// TwinCAT 3 PLC project Plc
// ProgramVersion: 3.1.4024.0
// libraries:
//   CHALET_BaseComponents, * (Beckhoff CH)
//   CHALET_Nc, * (Beckhoff CH)
//   CHALET_Xts, * (Beckhoff CH)
//   Tc2_ControllerToolbox, * (Beckhoff Automation GmbH)
//   Tc2_MC2, * (Beckhoff Automation GmbH)
//   Tc2_NC, * (Beckhoff Automation GmbH)
//   Tc2_Standard, * (Beckhoff Automation GmbH)
//   Tc2_System, * (Beckhoff Automation GmbH)
//   Tc3_Mc3Definitions, * (Beckhoff Automation GmbH)
//   Tc3_Module, * (Beckhoff Automation GmbH)
//   VisuDialogs, * (System)
//   VisuSymbols,newest,System
// project tree:
//   / GlobalTextList.TcGTLO, PlcTask.TcTTO, Visualisierungsmanager.TcVMO (not stored)
//   POUs/Example Product Data/ FB_ProductDataA.TcPOU, I_ProductDataA.TcIO (not stored), PRG_Example_ProductData.TcPOU, ST_ProductDataA.TcDUT (not stored)
//   POUs/Example Station Implementation/ E_StationProcessState.TcDUT, FB_StationBase.TcPOU, FB_StationLoadProcess.TcPOU, FB_StationUnLoadProcess.TcPOU, FB_StationMoutingProcess.TcPOU, I_StationProcess.TcIO, FB_StationCalibProcess.TcPOU, E_OpMode.TcDUT, PRG_Example_Station.TcPOU
//   POUs/ MAIN.TcPOU
//   VISUs/ Visualization.TcVIS
// real-time tasks:
//   TASK Task_Xts: cycle T#250us, priority 1, ADS port 350
//   TASK Task_Job: cycle default, priority 32
//   TASK Task_Plc: cycle T#10ms, priority 20, ADS port 351
// motion (NC):
//   TASK NC-Task 1 SAF: cycle T#2ms, priority 5, ADS port 501
//   TASK NC-Task 1 SVB: cycle T#10ms, priority 9, ADS port 511
//   AXIS Mover Axis 1 (id 1)
//     Dynamic: AccelerationMaximum=80000, DecelerationMaximum=80000, Acceleration=20000, Deceleration=20000, Jerk=200000
//     Velo: Maximum=4000
//     PositionAreaControl: Enable=false
//     TargetPosControl: Enable=false
//     OtherSettings: AllowMotionCmdToSlave=true, AllowMotionCmdToExtSetGenAxis=true
//     encoder EncType=28
//       EncPara: ModuloFactor=3000, ToleranceWndModuloStart=0.2, MaxCount=#xffffffff
//         ActPosCorrection: Enable=true, Time=0.1
//     drive DrvType=22
//       DrvPara: MaxCount=#xffffffff, DriveControlDWord=#x00000100
//         Analog: VeloReferenz=4200, TorqueSetpointScale=10
//         TimeComp: TaskDelayCycles=1
//     controller CtrType=1
//       CtrPara: PriorControlFactor=1
//         PosDiffControl: Range=10
//         Observer: BandWidth=20
//   AXIS Mover Axis 2 (id 2)
//     Dynamic: AccelerationMaximum=80000, DecelerationMaximum=80000, Acceleration=20000, Deceleration=20000, Jerk=200000
//     Velo: Maximum=4000
//     PositionAreaControl: Enable=false
//     TargetPosControl: Enable=false
//     OtherSettings: AllowMotionCmdToSlave=true, AllowMotionCmdToExtSetGenAxis=true
//     encoder EncType=28
//       EncPara: ModuloFactor=3000, ToleranceWndModuloStart=0.2, MaxCount=#xffffffff
//         ActPosCorrection: Enable=true, Time=0.1
//     drive DrvType=22
//       DrvPara: MaxCount=#xffffffff, DriveControlDWord=#x00000100
//         Analog: VeloReferenz=4200, TorqueSetpointScale=10
//         TimeComp: TaskDelayCycles=1
//     controller CtrType=1
//       CtrPara: PriorControlFactor=1
//         PosDiffControl: Range=10
//         Observer: BandWidth=20
//   AXIS Mover Axis 3 (id 3)
//     Dynamic: AccelerationMaximum=80000, DecelerationMaximum=80000, Acceleration=20000, Deceleration=20000, Jerk=200000
//     Velo: Maximum=4000
//     PositionAreaControl: Enable=false
//     TargetPosControl: Enable=false
//     OtherSettings: AllowMotionCmdToSlave=true, AllowMotionCmdToExtSetGenAxis=true
//     encoder EncType=28
//       EncPara: ModuloFactor=3000, ToleranceWndModuloStart=0.2, MaxCount=#xffffffff
//         ActPosCorrection: Enable=true, Time=0.1
//     drive DrvType=22
//       DrvPara: MaxCount=#xffffffff, DriveControlDWord=#x00000100
//         Analog: VeloReferenz=4200, TorqueSetpointScale=10
//         TimeComp: TaskDelayCycles=1
//     controller CtrType=1
//       CtrPara: PriorControlFactor=1
//         PosDiffControl: Range=10
//         Observer: BandWidth=20
//   AXIS Mover Axis 4 (id 4)
//     Dynamic: AccelerationMaximum=80000, DecelerationMaximum=80000, Acceleration=20000, Deceleration=20000, Jerk=200000
//     Velo: Maximum=4000
//     PositionAreaControl: Enable=false
//     TargetPosControl: Enable=false
//     OtherSettings: AllowMotionCmdToSlave=true, AllowMotionCmdToExtSetGenAxis=true
//     encoder EncType=28
//       EncPara: ModuloFactor=3000, ToleranceWndModuloStart=0.2, MaxCount=#xffffffff
//         ActPosCorrection: Enable=true, Time=0.1
//     drive DrvType=22
//       DrvPara: MaxCount=#xffffffff, DriveControlDWord=#x00000100
//         Analog: VeloReferenz=4200, TorqueSetpointScale=10
//         TimeComp: TaskDelayCycles=1
//     controller CtrType=1
//       CtrPara: PriorControlFactor=1
//         PosDiffControl: Range=10
//         Observer: BandWidth=20
//   AXIS Mover Axis 5 (id 5)
//     Dynamic: AccelerationMaximum=80000, DecelerationMaximum=80000, Acceleration=20000, Deceleration=20000, Jerk=200000
//     Velo: Maximum=4000
//     PositionAreaControl: Enable=false
//     TargetPosControl: Enable=false
//     OtherSettings: AllowMotionCmdToSlave=true, AllowMotionCmdToExtSetGenAxis=true
//     encoder EncType=28
//       EncPara: ModuloFactor=3000, ToleranceWndModuloStart=0.2, MaxCount=#xffffffff
//         ActPosCorrection: Enable=true, Time=0.1
//     drive DrvType=22
//       DrvPara: MaxCount=#xffffffff, DriveControlDWord=#x00000100
//         Analog: VeloReferenz=4200, TorqueSetpointScale=10
//         TimeComp: TaskDelayCycles=1
//     controller CtrType=1
//       CtrPara: PriorControlFactor=1
//         PosDiffControl: Range=10
//         Observer: BandWidth=20
//   AXIS Mover Axis 6 (id 6)
//     Dynamic: AccelerationMaximum=80000, DecelerationMaximum=80000, Acceleration=20000, Deceleration=20000, Jerk=200000
//     Velo: Maximum=4000
//     PositionAreaControl: Enable=false
//     TargetPosControl: Enable=false
//     OtherSettings: AllowMotionCmdToSlave=true, AllowMotionCmdToExtSetGenAxis=true
//     encoder EncType=28
//       EncPara: ModuloFactor=3000, ToleranceWndModuloStart=0.2, MaxCount=#xffffffff
//         ActPosCorrection: Enable=true, Time=0.1
//     drive DrvType=22
//       DrvPara: MaxCount=#xffffffff, DriveControlDWord=#x00000100
//         Analog: VeloReferenz=4200, TorqueSetpointScale=10
//         TimeComp: TaskDelayCycles=1
//     controller CtrType=1
//       CtrPara: PriorControlFactor=1
//         PosDiffControl: Range=10
//         Observer: BandWidth=20
//   AXIS Mover Axis 7 (id 7)
//     Dynamic: AccelerationMaximum=80000, DecelerationMaximum=80000, Acceleration=20000, Deceleration=20000, Jerk=200000
//     Velo: Maximum=4000
//     PositionAreaControl: Enable=false
//     TargetPosControl: Enable=false
//     OtherSettings: AllowMotionCmdToSlave=true, AllowMotionCmdToExtSetGenAxis=true
//     encoder EncType=28
//       EncPara: ModuloFactor=3000, ToleranceWndModuloStart=0.2, MaxCount=#xffffffff
//         ActPosCorrection: Enable=true, Time=0.1
//     drive DrvType=22
//       DrvPara: MaxCount=#xffffffff, DriveControlDWord=#x00000100
//         Analog: VeloReferenz=4200, TorqueSetpointScale=10
//         TimeComp: TaskDelayCycles=1
//     controller CtrType=1
//       CtrPara: PriorControlFactor=1
//         PosDiffControl: Range=10
//         Observer: BandWidth=20
//   AXIS Mover Axis 8 (id 8)
//     Dynamic: AccelerationMaximum=80000, DecelerationMaximum=80000, Acceleration=20000, Deceleration=20000, Jerk=200000
//     Velo: Maximum=4000
//     PositionAreaControl: Enable=false
//     TargetPosControl: Enable=false
//     OtherSettings: AllowMotionCmdToSlave=true, AllowMotionCmdToExtSetGenAxis=true
//     encoder EncType=28
//       EncPara: ModuloFactor=3000, ToleranceWndModuloStart=0.2, MaxCount=#xffffffff
//         ActPosCorrection: Enable=true, Time=0.1
//     drive DrvType=22
//       DrvPara: MaxCount=#xffffffff, DriveControlDWord=#x00000100
//         Analog: VeloReferenz=4200, TorqueSetpointScale=10
//         TimeComp: TaskDelayCycles=1
//     controller CtrType=1
//       CtrPara: PriorControlFactor=1
//         PosDiffControl: Range=10
//         Observer: BandWidth=20
//   AXIS SimAxis (id 9)
//     OtherSettings: AllowMotionCmdToSlave=true
//     encoder EncType=1
//     drive DrvType=5
//       Analog: TorqueSetpointScale=10, ScaleFactorActTorque=0.1
//       TimeComp: TaskDelayCycles=1
//     controller CtrType=1
//       CtrPara: PriorControlFactor=1
//         Observer: BandWidth=20
// I/O:
//   DEVICE Device 1 (RT-Ethernet Adapter)
//   DEVICE Device 5 (EtherCAT), AmsNetId 10.19.0.38.6.1
//     Box 1 (CU2508) [CU2508 Ethernet Port]
//     Term 2 (AT2001-0250) [AT2001-0250 Motor module with feed 250 mm, 48V]
//       Term 3 (AT2001-5250) [AT2001-5250 Sensor line with feed]
//     Term 4 (AT2000-0250) [AT2000-0250 Motor module 250 mm, 48V]
//       Term 5 (AT2000-5250) [AT2000-5250 Sensor line]
//     Term 6 (AT2000-0250) [AT2000-0250 Motor module 250 mm, 48V]
//       Term 7 (AT2000-5250) [AT2000-5250 Sensor line]
//   DEVICE Device 6 (EtherCAT), AmsNetId 10.19.0.38.7.1
//     Box 8 (CU2508) [CU2508 Ethernet Port]
//     Term 9 (AT2001-0250) [AT2001-0250 Motor module with feed 250 mm, 48V]
//       Term 10 (AT2001-5250) [AT2001-5250 Sensor line with feed]
//     Term 11 (AT2050-0500) [AT2050-0500 Motor module, 90° clothoid, EtherCAT In, 48V]
//       Term 12 (AT2050-5500) [AT2050-5500 Sensor line 90° clothoid, EtherCAT In]
//     Term 13 (AT2050-0501) [AT2050-0501 Motor module, 90° clothoid, EtherCAT Out, 48V]
//       Term 14 (AT2050-5501) [AT2050-5501 Sensor line 90° clothoid, EtherCAT Out]
//   DEVICE Device 7 (EtherCAT), AmsNetId 10.19.0.38.8.1
//     Box 15 (CU2508) [CU2508 Ethernet Port]
//     Term 16 (AT2001-0250) [AT2001-0250 Motor module with feed 250 mm, 48V]
//       Term 17 (AT2001-5250) [AT2001-5250 Sensor line with feed]
//     Term 18 (AT2000-0250) [AT2000-0250 Motor module 250 mm, 48V]
//       Term 19 (AT2000-5250) [AT2000-5250 Sensor line]
//     Term 20 (AT2000-0250) [AT2000-0250 Motor module 250 mm, 48V]
//       Term 21 (AT2000-5250) [AT2000-5250 Sensor line]
//   DEVICE Device 8 (EtherCAT), AmsNetId 10.19.0.38.9.1
//     Box 22 (CU2508) [CU2508 Ethernet Port]
//     Term 23 (AT2001-0250) [AT2001-0250 Motor module with feed 250 mm, 48V]
//       Term 24 (AT2001-5250) [AT2001-5250 Sensor line with feed]
//     Term 25 (AT2050-0500) [AT2050-0500 Motor module, 90° clothoid, EtherCAT In, 48V]
//       Term 26 (AT2050-5500) [AT2050-5500 Sensor line 90° clothoid, EtherCAT In]
//     Term 27 (AT2050-0501) [AT2050-0501 Motor module, 90° clothoid, EtherCAT Out, 48V]
//       Term 28 (AT2050-5501) [AT2050-5501 Sensor line 90° clothoid, EtherCAT Out]
//   DEVICE Gerät 3 (EtherCAT), AmsNetId 10.0.2.15.4.1
//     Klemme 36 (EK1100) [EK1100 EtherCAT-Koppler (2A E-Bus)]
//       Klemme 37 (EL6224) [EL6224 (IO Link Master)]
//       Klemme 3 (EL9011) [EL9011 Endklemme]
// variable links:
//   Device 5 (EtherCAT) <-> TcCOM Objects/XtsProcessingUnit 1/Part 1/Module 1
//     Term 2 (AT2001-0250)/CC Inputs/Current actual value Ch.1 <-> Data Pointer/CurrentActualValues[0]
//     Term 2 (AT2001-0250)/CC Inputs/Current actual value Ch.10 <-> Data Pointer/CurrentActualValues[9]
//     Term 2 (AT2001-0250)/CC Inputs/Current actual value Ch.11 <-> Data Pointer/CurrentActualValues[10]
//     Term 2 (AT2001-0250)/CC Inputs/Current actual value Ch.12 <-> Data Pointer/CurrentActualValues[11]
//     Term 2 (AT2001-0250)/CC Inputs/Current actual value Ch.13 <-> Data Pointer/CurrentActualValues[12]
//     Term 2 (AT2001-0250)/CC Inputs/Current actual value Ch.14 <-> Data Pointer/CurrentActualValues[13]
//     Term 2 (AT2001-0250)/CC Inputs/Current actual value Ch.15 <-> Data Pointer/CurrentActualValues[14]
//     Term 2 (AT2001-0250)/CC Inputs/Current actual value Ch.2 <-> Data Pointer/CurrentActualValues[1]
//     Term 2 (AT2001-0250)/CC Inputs/Current actual value Ch.3 <-> Data Pointer/CurrentActualValues[2]
//     Term 2 (AT2001-0250)/CC Inputs/Current actual value Ch.4 <-> Data Pointer/CurrentActualValues[3]
//     Term 2 (AT2001-0250)/CC Inputs/Current actual value Ch.5 <-> Data Pointer/CurrentActualValues[4]
//     Term 2 (AT2001-0250)/CC Inputs/Current actual value Ch.6 <-> Data Pointer/CurrentActualValues[5]
//     Term 2 (AT2001-0250)/CC Inputs/Current actual value Ch.7 <-> Data Pointer/CurrentActualValues[6]
//     Term 2 (AT2001-0250)/CC Inputs/Current actual value Ch.8 <-> Data Pointer/CurrentActualValues[7]
//     Term 2 (AT2001-0250)/CC Inputs/Current actual value Ch.9 <-> Data Pointer/CurrentActualValues[8]
//     Term 2 (AT2001-0250)/CC Inputs/Status <-> Data Pointer/Status
//     Term 2 (AT2001-0250)/CC Outputs/Control <-> Data Pointer/Control
//     Term 2 (AT2001-0250)/CC Outputs/Current setpoint value Ch.1 <-> Data Pointer/CurrentSetpointValues[0]
//     Term 2 (AT2001-0250)/CC Outputs/Current setpoint value Ch.10 <-> Data Pointer/CurrentSetpointValues[9]
//     Term 2 (AT2001-0250)/CC Outputs/Current setpoint value Ch.11 <-> Data Pointer/CurrentSetpointValues[10]
//     Term 2 (AT2001-0250)/CC Outputs/Current setpoint value Ch.12 <-> Data Pointer/CurrentSetpointValues[11]
//     Term 2 (AT2001-0250)/CC Outputs/Current setpoint value Ch.13 <-> Data Pointer/CurrentSetpointValues[12]
//     Term 2 (AT2001-0250)/CC Outputs/Current setpoint value Ch.14 <-> Data Pointer/CurrentSetpointValues[13]
//     Term 2 (AT2001-0250)/CC Outputs/Current setpoint value Ch.15 <-> Data Pointer/CurrentSetpointValues[14]
//     Term 2 (AT2001-0250)/CC Outputs/Current setpoint value Ch.2 <-> Data Pointer/CurrentSetpointValues[1]
//     Term 2 (AT2001-0250)/CC Outputs/Current setpoint value Ch.3 <-> Data Pointer/CurrentSetpointValues[2]
//     Term 2 (AT2001-0250)/CC Outputs/Current setpoint value Ch.4 <-> Data Pointer/CurrentSetpointValues[3]
//     Term 2 (AT2001-0250)/CC Outputs/Current setpoint value Ch.5 <-> Data Pointer/CurrentSetpointValues[4]
//     Term 2 (AT2001-0250)/CC Outputs/Current setpoint value Ch.6 <-> Data Pointer/CurrentSetpointValues[5]
//     Term 2 (AT2001-0250)/CC Outputs/Current setpoint value Ch.7 <-> Data Pointer/CurrentSetpointValues[6]
//     Term 2 (AT2001-0250)/CC Outputs/Current setpoint value Ch.8 <-> Data Pointer/CurrentSetpointValues[7]
//     Term 2 (AT2001-0250)/CC Outputs/Current setpoint value Ch.9 <-> Data Pointer/CurrentSetpointValues[8]
//     Term 2 (AT2001-0250)/Term 3 (AT2001-5250)/FB Inputs/Value Channel 01 <-> Data Pointer/RawPositionValues[0]
//     Term 2 (AT2001-0250)/Term 3 (AT2001-5250)/FB Inputs/Value Channel 02 <-> Data Pointer/RawPositionValues[1]
//     Term 2 (AT2001-0250)/Term 3 (AT2001-5250)/FB Inputs/Value Channel 03 <-> Data Pointer/RawPositionValues[2]
//     Term 2 (AT2001-0250)/Term 3 (AT2001-5250)/FB Inputs/Value Channel 04 <-> Data Pointer/RawPositionValues[3]
//     Term 2 (AT2001-0250)/Term 3 (AT2001-5250)/FB Inputs/Value Channel 05 <-> Data Pointer/RawPositionValues[4]
//     Term 2 (AT2001-0250)/Term 3 (AT2001-5250)/FB Inputs/Value Channel 06 <-> Data Pointer/RawPositionValues[5]
//     Term 2 (AT2001-0250)/Term 3 (AT2001-5250)/FB Inputs/Value Channel 07 <-> Data Pointer/RawPositionValues[6]
//     Term 2 (AT2001-0250)/Term 3 (AT2001-5250)/FB Inputs/Value Channel 08 <-> Data Pointer/RawPositionValues[7]
//     Term 2 (AT2001-0250)/Term 3 (AT2001-5250)/FB Inputs/Value Channel 09 <-> Data Pointer/RawPositionValues[8]
//     Term 2 (AT2001-0250)/Term 3 (AT2001-5250)/FB Inputs/Value Channel 10 <-> Data Pointer/RawPositionValues[9]
//     Term 2 (AT2001-0250)/Term 3 (AT2001-5250)/FB Inputs/Value Channel 11 <-> Data Pointer/RawPositionValues[10]
//     Term 2 (AT2001-0250)/Term 3 (AT2001-5250)/FB Inputs/Value Channel 12 <-> Data Pointer/RawPositionValues[11]
//     Term 2 (AT2001-0250)/Term 3 (AT2001-5250)/FB Inputs/Value Channel 13 <-> Data Pointer/RawPositionValues[12]
//     Term 2 (AT2001-0250)/Term 3 (AT2001-5250)/FB Inputs/Value Channel 14 <-> Data Pointer/RawPositionValues[13]
//     Term 2 (AT2001-0250)/Term 3 (AT2001-5250)/FB Inputs/Value Channel 15 <-> Data Pointer/RawPositionValues[14]
//     Term 2 (AT2001-0250)/Term 3 (AT2001-5250)/FB Inputs/Value Channel 16 <-> Data Pointer/RawPositionValues[15]
//     Term 2 (AT2001-0250)/Term 3 (AT2001-5250)/FB Inputs/Value Channel 17 <-> Data Pointer/RawPositionValues[16]
//     Term 2 (AT2001-0250)/Term 3 (AT2001-5250)/FB Inputs/Value Channel 18 <-> Data Pointer/RawPositionValues[17]
//     Term 2 (AT2001-0250)/Term 3 (AT2001-5250)/FB Inputs/Value Channel 19 <-> Data Pointer/RawPositionValues[18]
//     Term 2 (AT2001-0250)/Term 3 (AT2001-5250)/FB Inputs/Value Channel 20 <-> Data Pointer/RawPositionValues[19]
//     Term 2 (AT2001-0250)/Term 3 (AT2001-5250)/FB Inputs/Value Channel 21 <-> Data Pointer/RawPositionValues[20]
//     Term 2 (AT2001-0250)/Term 3 (AT2001-5250)/FB Inputs/Value Channel 22 <-> Data Pointer/RawPositionValues[21]
//     Term 2 (AT2001-0250)/Term 3 (AT2001-5250)/FB Inputs/Value Channel 23 <-> Data Pointer/RawPositionValues[22]
//     Term 2 (AT2001-0250)/Term 3 (AT2001-5250)/FB Inputs/Value Channel 24 <-> Data Pointer/RawPositionValues[23]
//     Term 2 (AT2001-0250)/Term 3 (AT2001-5250)/FB Inputs/Value Channel 25 <-> Data Pointer/RawPositionValues[24]
//     Term 2 (AT2001-0250)/Term 3 (AT2001-5250)/FB Inputs/Value Channel 26 <-> Data Pointer/RawPositionValues[25]
//     Term 2 (AT2001-0250)/Term 3 (AT2001-5250)/FB Inputs/Value Channel 27 <-> Data Pointer/RawPositionValues[26]
//     Term 2 (AT2001-0250)/Term 3 (AT2001-5250)/FB Inputs/Value Channel 28 <-> Data Pointer/RawPositionValues[27]
//     Term 2 (AT2001-0250)/Term 3 (AT2001-5250)/FB Inputs/Value Channel 29 <-> Data Pointer/RawPositionValues[28]
//     Term 2 (AT2001-0250)/Term 3 (AT2001-5250)/FB Inputs/Value Channel 30 <-> Data Pointer/RawPositionValues[29]
//     Term 2 (AT2001-0250)/Term 3 (AT2001-5250)/FB Inputs/Value Channel 31 <-> Data Pointer/RawPositionValues[30]
//     Term 2 (AT2001-0250)/Term 3 (AT2001-5250)/FB Inputs/Value Channel 32 <-> Data Pointer/RawPositionValues[31]
//   Device 5 (EtherCAT) <-> TcCOM Objects/XtsProcessingUnit 1/Part 1/Module 2
//     Term 4 (AT2000-0250)/CC Inputs/Current actual value Ch.1 <-> Data Pointer/CurrentActualValues[0]
//     Term 4 (AT2000-0250)/CC Inputs/Current actual value Ch.10 <-> Data Pointer/CurrentActualValues[9]
//     Term 4 (AT2000-0250)/CC Inputs/Current actual value Ch.11 <-> Data Pointer/CurrentActualValues[10]
//     Term 4 (AT2000-0250)/CC Inputs/Current actual value Ch.12 <-> Data Pointer/CurrentActualValues[11]
//     Term 4 (AT2000-0250)/CC Inputs/Current actual value Ch.13 <-> Data Pointer/CurrentActualValues[12]
//     Term 4 (AT2000-0250)/CC Inputs/Current actual value Ch.14 <-> Data Pointer/CurrentActualValues[13]
//     Term 4 (AT2000-0250)/CC Inputs/Current actual value Ch.15 <-> Data Pointer/CurrentActualValues[14]
//     Term 4 (AT2000-0250)/CC Inputs/Current actual value Ch.2 <-> Data Pointer/CurrentActualValues[1]
//     Term 4 (AT2000-0250)/CC Inputs/Current actual value Ch.3 <-> Data Pointer/CurrentActualValues[2]
//     Term 4 (AT2000-0250)/CC Inputs/Current actual value Ch.4 <-> Data Pointer/CurrentActualValues[3]
//     Term 4 (AT2000-0250)/CC Inputs/Current actual value Ch.5 <-> Data Pointer/CurrentActualValues[4]
//     Term 4 (AT2000-0250)/CC Inputs/Current actual value Ch.6 <-> Data Pointer/CurrentActualValues[5]
//     Term 4 (AT2000-0250)/CC Inputs/Current actual value Ch.7 <-> Data Pointer/CurrentActualValues[6]
//     Term 4 (AT2000-0250)/CC Inputs/Current actual value Ch.8 <-> Data Pointer/CurrentActualValues[7]
//     Term 4 (AT2000-0250)/CC Inputs/Current actual value Ch.9 <-> Data Pointer/CurrentActualValues[8]
//     Term 4 (AT2000-0250)/CC Inputs/Status <-> Data Pointer/Status
//     Term 4 (AT2000-0250)/CC Outputs/Control <-> Data Pointer/Control
//     Term 4 (AT2000-0250)/CC Outputs/Current setpoint value Ch.1 <-> Data Pointer/CurrentSetpointValues[0]
//     Term 4 (AT2000-0250)/CC Outputs/Current setpoint value Ch.10 <-> Data Pointer/CurrentSetpointValues[9]
//     Term 4 (AT2000-0250)/CC Outputs/Current setpoint value Ch.11 <-> Data Pointer/CurrentSetpointValues[10]
//     Term 4 (AT2000-0250)/CC Outputs/Current setpoint value Ch.12 <-> Data Pointer/CurrentSetpointValues[11]
//     Term 4 (AT2000-0250)/CC Outputs/Current setpoint value Ch.13 <-> Data Pointer/CurrentSetpointValues[12]
//     Term 4 (AT2000-0250)/CC Outputs/Current setpoint value Ch.14 <-> Data Pointer/CurrentSetpointValues[13]
//     Term 4 (AT2000-0250)/CC Outputs/Current setpoint value Ch.15 <-> Data Pointer/CurrentSetpointValues[14]
//     Term 4 (AT2000-0250)/CC Outputs/Current setpoint value Ch.2 <-> Data Pointer/CurrentSetpointValues[1]
//     Term 4 (AT2000-0250)/CC Outputs/Current setpoint value Ch.3 <-> Data Pointer/CurrentSetpointValues[2]
//     Term 4 (AT2000-0250)/CC Outputs/Current setpoint value Ch.4 <-> Data Pointer/CurrentSetpointValues[3]
//     Term 4 (AT2000-0250)/CC Outputs/Current setpoint value Ch.5 <-> Data Pointer/CurrentSetpointValues[4]
//     Term 4 (AT2000-0250)/CC Outputs/Current setpoint value Ch.6 <-> Data Pointer/CurrentSetpointValues[5]
//     Term 4 (AT2000-0250)/CC Outputs/Current setpoint value Ch.7 <-> Data Pointer/CurrentSetpointValues[6]
//     Term 4 (AT2000-0250)/CC Outputs/Current setpoint value Ch.8 <-> Data Pointer/CurrentSetpointValues[7]
//     Term 4 (AT2000-0250)/CC Outputs/Current setpoint value Ch.9 <-> Data Pointer/CurrentSetpointValues[8]
//     Term 4 (AT2000-0250)/Term 5 (AT2000-5250)/FB Inputs/Value Channel 01 <-> Data Pointer/RawPositionValues[0]
//     Term 4 (AT2000-0250)/Term 5 (AT2000-5250)/FB Inputs/Value Channel 02 <-> Data Pointer/RawPositionValues[1]
//     Term 4 (AT2000-0250)/Term 5 (AT2000-5250)/FB Inputs/Value Channel 03 <-> Data Pointer/RawPositionValues[2]
//     Term 4 (AT2000-0250)/Term 5 (AT2000-5250)/FB Inputs/Value Channel 04 <-> Data Pointer/RawPositionValues[3]
//     Term 4 (AT2000-0250)/Term 5 (AT2000-5250)/FB Inputs/Value Channel 05 <-> Data Pointer/RawPositionValues[4]
//     Term 4 (AT2000-0250)/Term 5 (AT2000-5250)/FB Inputs/Value Channel 06 <-> Data Pointer/RawPositionValues[5]
//     Term 4 (AT2000-0250)/Term 5 (AT2000-5250)/FB Inputs/Value Channel 07 <-> Data Pointer/RawPositionValues[6]
//     Term 4 (AT2000-0250)/Term 5 (AT2000-5250)/FB Inputs/Value Channel 08 <-> Data Pointer/RawPositionValues[7]
//     Term 4 (AT2000-0250)/Term 5 (AT2000-5250)/FB Inputs/Value Channel 09 <-> Data Pointer/RawPositionValues[8]
//     Term 4 (AT2000-0250)/Term 5 (AT2000-5250)/FB Inputs/Value Channel 10 <-> Data Pointer/RawPositionValues[9]
//     Term 4 (AT2000-0250)/Term 5 (AT2000-5250)/FB Inputs/Value Channel 11 <-> Data Pointer/RawPositionValues[10]
//     Term 4 (AT2000-0250)/Term 5 (AT2000-5250)/FB Inputs/Value Channel 12 <-> Data Pointer/RawPositionValues[11]
//     Term 4 (AT2000-0250)/Term 5 (AT2000-5250)/FB Inputs/Value Channel 13 <-> Data Pointer/RawPositionValues[12]
//     Term 4 (AT2000-0250)/Term 5 (AT2000-5250)/FB Inputs/Value Channel 14 <-> Data Pointer/RawPositionValues[13]
//     Term 4 (AT2000-0250)/Term 5 (AT2000-5250)/FB Inputs/Value Channel 15 <-> Data Pointer/RawPositionValues[14]
//     Term 4 (AT2000-0250)/Term 5 (AT2000-5250)/FB Inputs/Value Channel 16 <-> Data Pointer/RawPositionValues[15]
//     Term 4 (AT2000-0250)/Term 5 (AT2000-5250)/FB Inputs/Value Channel 17 <-> Data Pointer/RawPositionValues[16]
//     Term 4 (AT2000-0250)/Term 5 (AT2000-5250)/FB Inputs/Value Channel 18 <-> Data Pointer/RawPositionValues[17]
//     Term 4 (AT2000-0250)/Term 5 (AT2000-5250)/FB Inputs/Value Channel 19 <-> Data Pointer/RawPositionValues[18]
//     Term 4 (AT2000-0250)/Term 5 (AT2000-5250)/FB Inputs/Value Channel 20 <-> Data Pointer/RawPositionValues[19]
//     Term 4 (AT2000-0250)/Term 5 (AT2000-5250)/FB Inputs/Value Channel 21 <-> Data Pointer/RawPositionValues[20]
//     Term 4 (AT2000-0250)/Term 5 (AT2000-5250)/FB Inputs/Value Channel 22 <-> Data Pointer/RawPositionValues[21]
//     Term 4 (AT2000-0250)/Term 5 (AT2000-5250)/FB Inputs/Value Channel 23 <-> Data Pointer/RawPositionValues[22]
//     Term 4 (AT2000-0250)/Term 5 (AT2000-5250)/FB Inputs/Value Channel 24 <-> Data Pointer/RawPositionValues[23]
//     Term 4 (AT2000-0250)/Term 5 (AT2000-5250)/FB Inputs/Value Channel 25 <-> Data Pointer/RawPositionValues[24]
//     Term 4 (AT2000-0250)/Term 5 (AT2000-5250)/FB Inputs/Value Channel 26 <-> Data Pointer/RawPositionValues[25]
//     Term 4 (AT2000-0250)/Term 5 (AT2000-5250)/FB Inputs/Value Channel 27 <-> Data Pointer/RawPositionValues[26]
//     Term 4 (AT2000-0250)/Term 5 (AT2000-5250)/FB Inputs/Value Channel 28 <-> Data Pointer/RawPositionValues[27]
//     Term 4 (AT2000-0250)/Term 5 (AT2000-5250)/FB Inputs/Value Channel 29 <-> Data Pointer/RawPositionValues[28]
//     Term 4 (AT2000-0250)/Term 5 (AT2000-5250)/FB Inputs/Value Channel 30 <-> Data Pointer/RawPositionValues[29]
//     Term 4 (AT2000-0250)/Term 5 (AT2000-5250)/FB Inputs/Value Channel 31 <-> Data Pointer/RawPositionValues[30]
//     Term 4 (AT2000-0250)/Term 5 (AT2000-5250)/FB Inputs/Value Channel 32 <-> Data Pointer/RawPositionValues[31]
//   Device 5 (EtherCAT) <-> TcCOM Objects/XtsProcessingUnit 1/Part 1/Module 3
//     Term 6 (AT2000-0250)/CC Inputs/Current actual value Ch.1 <-> Data Pointer/CurrentActualValues[0]
//     Term 6 (AT2000-0250)/CC Inputs/Current actual value Ch.10 <-> Data Pointer/CurrentActualValues[9]
//     Term 6 (AT2000-0250)/CC Inputs/Current actual value Ch.11 <-> Data Pointer/CurrentActualValues[10]
//     Term 6 (AT2000-0250)/CC Inputs/Current actual value Ch.12 <-> Data Pointer/CurrentActualValues[11]
//     Term 6 (AT2000-0250)/CC Inputs/Current actual value Ch.13 <-> Data Pointer/CurrentActualValues[12]
//     Term 6 (AT2000-0250)/CC Inputs/Current actual value Ch.14 <-> Data Pointer/CurrentActualValues[13]
//     Term 6 (AT2000-0250)/CC Inputs/Current actual value Ch.15 <-> Data Pointer/CurrentActualValues[14]
//     Term 6 (AT2000-0250)/CC Inputs/Current actual value Ch.2 <-> Data Pointer/CurrentActualValues[1]
//     Term 6 (AT2000-0250)/CC Inputs/Current actual value Ch.3 <-> Data Pointer/CurrentActualValues[2]
//     Term 6 (AT2000-0250)/CC Inputs/Current actual value Ch.4 <-> Data Pointer/CurrentActualValues[3]
//     Term 6 (AT2000-0250)/CC Inputs/Current actual value Ch.5 <-> Data Pointer/CurrentActualValues[4]
//     Term 6 (AT2000-0250)/CC Inputs/Current actual value Ch.6 <-> Data Pointer/CurrentActualValues[5]
//     Term 6 (AT2000-0250)/CC Inputs/Current actual value Ch.7 <-> Data Pointer/CurrentActualValues[6]
//     Term 6 (AT2000-0250)/CC Inputs/Current actual value Ch.8 <-> Data Pointer/CurrentActualValues[7]
//     Term 6 (AT2000-0250)/CC Inputs/Current actual value Ch.9 <-> Data Pointer/CurrentActualValues[8]
//     Term 6 (AT2000-0250)/CC Inputs/Status <-> Data Pointer/Status
//     Term 6 (AT2000-0250)/CC Outputs/Control <-> Data Pointer/Control
//     Term 6 (AT2000-0250)/CC Outputs/Current setpoint value Ch.1 <-> Data Pointer/CurrentSetpointValues[0]
//     Term 6 (AT2000-0250)/CC Outputs/Current setpoint value Ch.10 <-> Data Pointer/CurrentSetpointValues[9]
//     Term 6 (AT2000-0250)/CC Outputs/Current setpoint value Ch.11 <-> Data Pointer/CurrentSetpointValues[10]
//     Term 6 (AT2000-0250)/CC Outputs/Current setpoint value Ch.12 <-> Data Pointer/CurrentSetpointValues[11]
//     Term 6 (AT2000-0250)/CC Outputs/Current setpoint value Ch.13 <-> Data Pointer/CurrentSetpointValues[12]
//     Term 6 (AT2000-0250)/CC Outputs/Current setpoint value Ch.14 <-> Data Pointer/CurrentSetpointValues[13]
//     Term 6 (AT2000-0250)/CC Outputs/Current setpoint value Ch.15 <-> Data Pointer/CurrentSetpointValues[14]
//     Term 6 (AT2000-0250)/CC Outputs/Current setpoint value Ch.2 <-> Data Pointer/CurrentSetpointValues[1]
//     Term 6 (AT2000-0250)/CC Outputs/Current setpoint value Ch.3 <-> Data Pointer/CurrentSetpointValues[2]
//     Term 6 (AT2000-0250)/CC Outputs/Current setpoint value Ch.4 <-> Data Pointer/CurrentSetpointValues[3]
//     Term 6 (AT2000-0250)/CC Outputs/Current setpoint value Ch.5 <-> Data Pointer/CurrentSetpointValues[4]
//     Term 6 (AT2000-0250)/CC Outputs/Current setpoint value Ch.6 <-> Data Pointer/CurrentSetpointValues[5]
//     Term 6 (AT2000-0250)/CC Outputs/Current setpoint value Ch.7 <-> Data Pointer/CurrentSetpointValues[6]
//     Term 6 (AT2000-0250)/CC Outputs/Current setpoint value Ch.8 <-> Data Pointer/CurrentSetpointValues[7]
//     Term 6 (AT2000-0250)/CC Outputs/Current setpoint value Ch.9 <-> Data Pointer/CurrentSetpointValues[8]
//     Term 6 (AT2000-0250)/Term 7 (AT2000-5250)/FB Inputs/Value Channel 01 <-> Data Pointer/RawPositionValues[0]
//     Term 6 (AT2000-0250)/Term 7 (AT2000-5250)/FB Inputs/Value Channel 02 <-> Data Pointer/RawPositionValues[1]
//     Term 6 (AT2000-0250)/Term 7 (AT2000-5250)/FB Inputs/Value Channel 03 <-> Data Pointer/RawPositionValues[2]
//     Term 6 (AT2000-0250)/Term 7 (AT2000-5250)/FB Inputs/Value Channel 04 <-> Data Pointer/RawPositionValues[3]
//     Term 6 (AT2000-0250)/Term 7 (AT2000-5250)/FB Inputs/Value Channel 05 <-> Data Pointer/RawPositionValues[4]
//     Term 6 (AT2000-0250)/Term 7 (AT2000-5250)/FB Inputs/Value Channel 06 <-> Data Pointer/RawPositionValues[5]
//     Term 6 (AT2000-0250)/Term 7 (AT2000-5250)/FB Inputs/Value Channel 07 <-> Data Pointer/RawPositionValues[6]
//     Term 6 (AT2000-0250)/Term 7 (AT2000-5250)/FB Inputs/Value Channel 08 <-> Data Pointer/RawPositionValues[7]
//     Term 6 (AT2000-0250)/Term 7 (AT2000-5250)/FB Inputs/Value Channel 09 <-> Data Pointer/RawPositionValues[8]
//     Term 6 (AT2000-0250)/Term 7 (AT2000-5250)/FB Inputs/Value Channel 10 <-> Data Pointer/RawPositionValues[9]
//     Term 6 (AT2000-0250)/Term 7 (AT2000-5250)/FB Inputs/Value Channel 11 <-> Data Pointer/RawPositionValues[10]
//     Term 6 (AT2000-0250)/Term 7 (AT2000-5250)/FB Inputs/Value Channel 12 <-> Data Pointer/RawPositionValues[11]
//     Term 6 (AT2000-0250)/Term 7 (AT2000-5250)/FB Inputs/Value Channel 13 <-> Data Pointer/RawPositionValues[12]
//     Term 6 (AT2000-0250)/Term 7 (AT2000-5250)/FB Inputs/Value Channel 14 <-> Data Pointer/RawPositionValues[13]
//     Term 6 (AT2000-0250)/Term 7 (AT2000-5250)/FB Inputs/Value Channel 15 <-> Data Pointer/RawPositionValues[14]
//     Term 6 (AT2000-0250)/Term 7 (AT2000-5250)/FB Inputs/Value Channel 16 <-> Data Pointer/RawPositionValues[15]
//     Term 6 (AT2000-0250)/Term 7 (AT2000-5250)/FB Inputs/Value Channel 17 <-> Data Pointer/RawPositionValues[16]
//     Term 6 (AT2000-0250)/Term 7 (AT2000-5250)/FB Inputs/Value Channel 18 <-> Data Pointer/RawPositionValues[17]
//     Term 6 (AT2000-0250)/Term 7 (AT2000-5250)/FB Inputs/Value Channel 19 <-> Data Pointer/RawPositionValues[18]
//     Term 6 (AT2000-0250)/Term 7 (AT2000-5250)/FB Inputs/Value Channel 20 <-> Data Pointer/RawPositionValues[19]
//     Term 6 (AT2000-0250)/Term 7 (AT2000-5250)/FB Inputs/Value Channel 21 <-> Data Pointer/RawPositionValues[20]
//     Term 6 (AT2000-0250)/Term 7 (AT2000-5250)/FB Inputs/Value Channel 22 <-> Data Pointer/RawPositionValues[21]
//     Term 6 (AT2000-0250)/Term 7 (AT2000-5250)/FB Inputs/Value Channel 23 <-> Data Pointer/RawPositionValues[22]
//     Term 6 (AT2000-0250)/Term 7 (AT2000-5250)/FB Inputs/Value Channel 24 <-> Data Pointer/RawPositionValues[23]
//     Term 6 (AT2000-0250)/Term 7 (AT2000-5250)/FB Inputs/Value Channel 25 <-> Data Pointer/RawPositionValues[24]
//     Term 6 (AT2000-0250)/Term 7 (AT2000-5250)/FB Inputs/Value Channel 26 <-> Data Pointer/RawPositionValues[25]
//     Term 6 (AT2000-0250)/Term 7 (AT2000-5250)/FB Inputs/Value Channel 27 <-> Data Pointer/RawPositionValues[26]
//     Term 6 (AT2000-0250)/Term 7 (AT2000-5250)/FB Inputs/Value Channel 28 <-> Data Pointer/RawPositionValues[27]
//     Term 6 (AT2000-0250)/Term 7 (AT2000-5250)/FB Inputs/Value Channel 29 <-> Data Pointer/RawPositionValues[28]
//     Term 6 (AT2000-0250)/Term 7 (AT2000-5250)/FB Inputs/Value Channel 30 <-> Data Pointer/RawPositionValues[29]
//     Term 6 (AT2000-0250)/Term 7 (AT2000-5250)/FB Inputs/Value Channel 31 <-> Data Pointer/RawPositionValues[30]
//     Term 6 (AT2000-0250)/Term 7 (AT2000-5250)/FB Inputs/Value Channel 32 <-> Data Pointer/RawPositionValues[31]
//   Device 6 (EtherCAT) <-> TcCOM Objects/XtsProcessingUnit 1/Part 1/Module 4
//     Term 9 (AT2001-0250)/CC Inputs/Current actual value Ch.1 <-> Data Pointer/CurrentActualValues[0]
//     Term 9 (AT2001-0250)/CC Inputs/Current actual value Ch.10 <-> Data Pointer/CurrentActualValues[9]
//     Term 9 (AT2001-0250)/CC Inputs/Current actual value Ch.11 <-> Data Pointer/CurrentActualValues[10]
//     Term 9 (AT2001-0250)/CC Inputs/Current actual value Ch.12 <-> Data Pointer/CurrentActualValues[11]
//     Term 9 (AT2001-0250)/CC Inputs/Current actual value Ch.13 <-> Data Pointer/CurrentActualValues[12]
//     Term 9 (AT2001-0250)/CC Inputs/Current actual value Ch.14 <-> Data Pointer/CurrentActualValues[13]
//     Term 9 (AT2001-0250)/CC Inputs/Current actual value Ch.15 <-> Data Pointer/CurrentActualValues[14]
//     Term 9 (AT2001-0250)/CC Inputs/Current actual value Ch.2 <-> Data Pointer/CurrentActualValues[1]
//     Term 9 (AT2001-0250)/CC Inputs/Current actual value Ch.3 <-> Data Pointer/CurrentActualValues[2]
//     Term 9 (AT2001-0250)/CC Inputs/Current actual value Ch.4 <-> Data Pointer/CurrentActualValues[3]
//     Term 9 (AT2001-0250)/CC Inputs/Current actual value Ch.5 <-> Data Pointer/CurrentActualValues[4]
//     Term 9 (AT2001-0250)/CC Inputs/Current actual value Ch.6 <-> Data Pointer/CurrentActualValues[5]
//     Term 9 (AT2001-0250)/CC Inputs/Current actual value Ch.7 <-> Data Pointer/CurrentActualValues[6]
//     Term 9 (AT2001-0250)/CC Inputs/Current actual value Ch.8 <-> Data Pointer/CurrentActualValues[7]
//     Term 9 (AT2001-0250)/CC Inputs/Current actual value Ch.9 <-> Data Pointer/CurrentActualValues[8]
//     Term 9 (AT2001-0250)/CC Inputs/Status <-> Data Pointer/Status
//     Term 9 (AT2001-0250)/CC Outputs/Control <-> Data Pointer/Control
//     Term 9 (AT2001-0250)/CC Outputs/Current setpoint value Ch.1 <-> Data Pointer/CurrentSetpointValues[0]
//     Term 9 (AT2001-0250)/CC Outputs/Current setpoint value Ch.10 <-> Data Pointer/CurrentSetpointValues[9]
//     Term 9 (AT2001-0250)/CC Outputs/Current setpoint value Ch.11 <-> Data Pointer/CurrentSetpointValues[10]
//     Term 9 (AT2001-0250)/CC Outputs/Current setpoint value Ch.12 <-> Data Pointer/CurrentSetpointValues[11]
//     Term 9 (AT2001-0250)/CC Outputs/Current setpoint value Ch.13 <-> Data Pointer/CurrentSetpointValues[12]
//     Term 9 (AT2001-0250)/CC Outputs/Current setpoint value Ch.14 <-> Data Pointer/CurrentSetpointValues[13]
//     Term 9 (AT2001-0250)/CC Outputs/Current setpoint value Ch.15 <-> Data Pointer/CurrentSetpointValues[14]
//     Term 9 (AT2001-0250)/CC Outputs/Current setpoint value Ch.2 <-> Data Pointer/CurrentSetpointValues[1]
//     Term 9 (AT2001-0250)/CC Outputs/Current setpoint value Ch.3 <-> Data Pointer/CurrentSetpointValues[2]
//     Term 9 (AT2001-0250)/CC Outputs/Current setpoint value Ch.4 <-> Data Pointer/CurrentSetpointValues[3]
//     Term 9 (AT2001-0250)/CC Outputs/Current setpoint value Ch.5 <-> Data Pointer/CurrentSetpointValues[4]
//     Term 9 (AT2001-0250)/CC Outputs/Current setpoint value Ch.6 <-> Data Pointer/CurrentSetpointValues[5]
//     Term 9 (AT2001-0250)/CC Outputs/Current setpoint value Ch.7 <-> Data Pointer/CurrentSetpointValues[6]
//     Term 9 (AT2001-0250)/CC Outputs/Current setpoint value Ch.8 <-> Data Pointer/CurrentSetpointValues[7]
//     Term 9 (AT2001-0250)/CC Outputs/Current setpoint value Ch.9 <-> Data Pointer/CurrentSetpointValues[8]
//     Term 9 (AT2001-0250)/Term 10 (AT2001-5250)/FB Inputs/Value Channel 01 <-> Data Pointer/RawPositionValues[0]
//     Term 9 (AT2001-0250)/Term 10 (AT2001-5250)/FB Inputs/Value Channel 02 <-> Data Pointer/RawPositionValues[1]
//     Term 9 (AT2001-0250)/Term 10 (AT2001-5250)/FB Inputs/Value Channel 03 <-> Data Pointer/RawPositionValues[2]
//     Term 9 (AT2001-0250)/Term 10 (AT2001-5250)/FB Inputs/Value Channel 04 <-> Data Pointer/RawPositionValues[3]
//     Term 9 (AT2001-0250)/Term 10 (AT2001-5250)/FB Inputs/Value Channel 05 <-> Data Pointer/RawPositionValues[4]
//     Term 9 (AT2001-0250)/Term 10 (AT2001-5250)/FB Inputs/Value Channel 06 <-> Data Pointer/RawPositionValues[5]
//     Term 9 (AT2001-0250)/Term 10 (AT2001-5250)/FB Inputs/Value Channel 07 <-> Data Pointer/RawPositionValues[6]
//     Term 9 (AT2001-0250)/Term 10 (AT2001-5250)/FB Inputs/Value Channel 08 <-> Data Pointer/RawPositionValues[7]
//     Term 9 (AT2001-0250)/Term 10 (AT2001-5250)/FB Inputs/Value Channel 09 <-> Data Pointer/RawPositionValues[8]
//     Term 9 (AT2001-0250)/Term 10 (AT2001-5250)/FB Inputs/Value Channel 10 <-> Data Pointer/RawPositionValues[9]
//     Term 9 (AT2001-0250)/Term 10 (AT2001-5250)/FB Inputs/Value Channel 11 <-> Data Pointer/RawPositionValues[10]
//     Term 9 (AT2001-0250)/Term 10 (AT2001-5250)/FB Inputs/Value Channel 12 <-> Data Pointer/RawPositionValues[11]
//     Term 9 (AT2001-0250)/Term 10 (AT2001-5250)/FB Inputs/Value Channel 13 <-> Data Pointer/RawPositionValues[12]
//     Term 9 (AT2001-0250)/Term 10 (AT2001-5250)/FB Inputs/Value Channel 14 <-> Data Pointer/RawPositionValues[13]
//     Term 9 (AT2001-0250)/Term 10 (AT2001-5250)/FB Inputs/Value Channel 15 <-> Data Pointer/RawPositionValues[14]
//     Term 9 (AT2001-0250)/Term 10 (AT2001-5250)/FB Inputs/Value Channel 16 <-> Data Pointer/RawPositionValues[15]
//     Term 9 (AT2001-0250)/Term 10 (AT2001-5250)/FB Inputs/Value Channel 17 <-> Data Pointer/RawPositionValues[16]
//     Term 9 (AT2001-0250)/Term 10 (AT2001-5250)/FB Inputs/Value Channel 18 <-> Data Pointer/RawPositionValues[17]
//     Term 9 (AT2001-0250)/Term 10 (AT2001-5250)/FB Inputs/Value Channel 19 <-> Data Pointer/RawPositionValues[18]
//     Term 9 (AT2001-0250)/Term 10 (AT2001-5250)/FB Inputs/Value Channel 20 <-> Data Pointer/RawPositionValues[19]
//     Term 9 (AT2001-0250)/Term 10 (AT2001-5250)/FB Inputs/Value Channel 21 <-> Data Pointer/RawPositionValues[20]
//     Term 9 (AT2001-0250)/Term 10 (AT2001-5250)/FB Inputs/Value Channel 22 <-> Data Pointer/RawPositionValues[21]
//     Term 9 (AT2001-0250)/Term 10 (AT2001-5250)/FB Inputs/Value Channel 23 <-> Data Pointer/RawPositionValues[22]
//     Term 9 (AT2001-0250)/Term 10 (AT2001-5250)/FB Inputs/Value Channel 24 <-> Data Pointer/RawPositionValues[23]
//     Term 9 (AT2001-0250)/Term 10 (AT2001-5250)/FB Inputs/Value Channel 25 <-> Data Pointer/RawPositionValues[24]
//     Term 9 (AT2001-0250)/Term 10 (AT2001-5250)/FB Inputs/Value Channel 26 <-> Data Pointer/RawPositionValues[25]
//     Term 9 (AT2001-0250)/Term 10 (AT2001-5250)/FB Inputs/Value Channel 27 <-> Data Pointer/RawPositionValues[26]
//     Term 9 (AT2001-0250)/Term 10 (AT2001-5250)/FB Inputs/Value Channel 28 <-> Data Pointer/RawPositionValues[27]
//     Term 9 (AT2001-0250)/Term 10 (AT2001-5250)/FB Inputs/Value Channel 29 <-> Data Pointer/RawPositionValues[28]
//     Term 9 (AT2001-0250)/Term 10 (AT2001-5250)/FB Inputs/Value Channel 30 <-> Data Pointer/RawPositionValues[29]
//     Term 9 (AT2001-0250)/Term 10 (AT2001-5250)/FB Inputs/Value Channel 31 <-> Data Pointer/RawPositionValues[30]
//     Term 9 (AT2001-0250)/Term 10 (AT2001-5250)/FB Inputs/Value Channel 32 <-> Data Pointer/RawPositionValues[31]
//   Device 6 (EtherCAT) <-> TcCOM Objects/XtsProcessingUnit 1/Part 1/Module 5
//     Term 11 (AT2050-0500)/CC Inputs/Current actual value Ch.1 <-> Data Pointer/CurrentActualValues[0]
//     Term 11 (AT2050-0500)/CC Inputs/Current actual value Ch.10 <-> Data Pointer/CurrentActualValues[9]
//     Term 11 (AT2050-0500)/CC Inputs/Current actual value Ch.11 <-> Data Pointer/CurrentActualValues[10]
//     Term 11 (AT2050-0500)/CC Inputs/Current actual value Ch.12 <-> Data Pointer/CurrentActualValues[11]
//     Term 11 (AT2050-0500)/CC Inputs/Current actual value Ch.13 <-> Data Pointer/CurrentActualValues[12]
//     Term 11 (AT2050-0500)/CC Inputs/Current actual value Ch.14 <-> Data Pointer/CurrentActualValues[13]
//     Term 11 (AT2050-0500)/CC Inputs/Current actual value Ch.15 <-> Data Pointer/CurrentActualValues[14]
//     Term 11 (AT2050-0500)/CC Inputs/Current actual value Ch.2 <-> Data Pointer/CurrentActualValues[1]
//     Term 11 (AT2050-0500)/CC Inputs/Current actual value Ch.3 <-> Data Pointer/CurrentActualValues[2]
//     Term 11 (AT2050-0500)/CC Inputs/Current actual value Ch.4 <-> Data Pointer/CurrentActualValues[3]
//     Term 11 (AT2050-0500)/CC Inputs/Current actual value Ch.5 <-> Data Pointer/CurrentActualValues[4]
//     Term 11 (AT2050-0500)/CC Inputs/Current actual value Ch.6 <-> Data Pointer/CurrentActualValues[5]
//     Term 11 (AT2050-0500)/CC Inputs/Current actual value Ch.7 <-> Data Pointer/CurrentActualValues[6]
//     Term 11 (AT2050-0500)/CC Inputs/Current actual value Ch.8 <-> Data Pointer/CurrentActualValues[7]
//     Term 11 (AT2050-0500)/CC Inputs/Current actual value Ch.9 <-> Data Pointer/CurrentActualValues[8]
//     Term 11 (AT2050-0500)/CC Inputs/Status <-> Data Pointer/Status
//     Term 11 (AT2050-0500)/CC Outputs/Control <-> Data Pointer/Control
//     Term 11 (AT2050-0500)/CC Outputs/Current setpoint value Ch.1 <-> Data Pointer/CurrentSetpointValues[0]
//     Term 11 (AT2050-0500)/CC Outputs/Current setpoint value Ch.10 <-> Data Pointer/CurrentSetpointValues[9]
//     Term 11 (AT2050-0500)/CC Outputs/Current setpoint value Ch.11 <-> Data Pointer/CurrentSetpointValues[10]
//     Term 11 (AT2050-0500)/CC Outputs/Current setpoint value Ch.12 <-> Data Pointer/CurrentSetpointValues[11]
//     Term 11 (AT2050-0500)/CC Outputs/Current setpoint value Ch.13 <-> Data Pointer/CurrentSetpointValues[12]
//     Term 11 (AT2050-0500)/CC Outputs/Current setpoint value Ch.14 <-> Data Pointer/CurrentSetpointValues[13]
//     Term 11 (AT2050-0500)/CC Outputs/Current setpoint value Ch.15 <-> Data Pointer/CurrentSetpointValues[14]
//     Term 11 (AT2050-0500)/CC Outputs/Current setpoint value Ch.2 <-> Data Pointer/CurrentSetpointValues[1]
//     Term 11 (AT2050-0500)/CC Outputs/Current setpoint value Ch.3 <-> Data Pointer/CurrentSetpointValues[2]
//     Term 11 (AT2050-0500)/CC Outputs/Current setpoint value Ch.4 <-> Data Pointer/CurrentSetpointValues[3]
//     Term 11 (AT2050-0500)/CC Outputs/Current setpoint value Ch.5 <-> Data Pointer/CurrentSetpointValues[4]
//     Term 11 (AT2050-0500)/CC Outputs/Current setpoint value Ch.6 <-> Data Pointer/CurrentSetpointValues[5]
//     Term 11 (AT2050-0500)/CC Outputs/Current setpoint value Ch.7 <-> Data Pointer/CurrentSetpointValues[6]
//     Term 11 (AT2050-0500)/CC Outputs/Current setpoint value Ch.8 <-> Data Pointer/CurrentSetpointValues[7]
//     Term 11 (AT2050-0500)/CC Outputs/Current setpoint value Ch.9 <-> Data Pointer/CurrentSetpointValues[8]
//     Term 11 (AT2050-0500)/Term 12 (AT2050-5500)/FB Inputs/Value Channel 01 <-> Data Pointer/RawPositionValues[0]
//     Term 11 (AT2050-0500)/Term 12 (AT2050-5500)/FB Inputs/Value Channel 02 <-> Data Pointer/RawPositionValues[1]
//     Term 11 (AT2050-0500)/Term 12 (AT2050-5500)/FB Inputs/Value Channel 03 <-> Data Pointer/RawPositionValues[2]
//     Term 11 (AT2050-0500)/Term 12 (AT2050-5500)/FB Inputs/Value Channel 04 <-> Data Pointer/RawPositionValues[3]
//     Term 11 (AT2050-0500)/Term 12 (AT2050-5500)/FB Inputs/Value Channel 05 <-> Data Pointer/RawPositionValues[4]
//     Term 11 (AT2050-0500)/Term 12 (AT2050-5500)/FB Inputs/Value Channel 06 <-> Data Pointer/RawPositionValues[5]
//     Term 11 (AT2050-0500)/Term 12 (AT2050-5500)/FB Inputs/Value Channel 07 <-> Data Pointer/RawPositionValues[6]
//     Term 11 (AT2050-0500)/Term 12 (AT2050-5500)/FB Inputs/Value Channel 08 <-> Data Pointer/RawPositionValues[7]
//     Term 11 (AT2050-0500)/Term 12 (AT2050-5500)/FB Inputs/Value Channel 09 <-> Data Pointer/RawPositionValues[8]
//     Term 11 (AT2050-0500)/Term 12 (AT2050-5500)/FB Inputs/Value Channel 10 <-> Data Pointer/RawPositionValues[9]
//     Term 11 (AT2050-0500)/Term 12 (AT2050-5500)/FB Inputs/Value Channel 11 <-> Data Pointer/RawPositionValues[10]
//     Term 11 (AT2050-0500)/Term 12 (AT2050-5500)/FB Inputs/Value Channel 12 <-> Data Pointer/RawPositionValues[11]
//     Term 11 (AT2050-0500)/Term 12 (AT2050-5500)/FB Inputs/Value Channel 13 <-> Data Pointer/RawPositionValues[12]
//     Term 11 (AT2050-0500)/Term 12 (AT2050-5500)/FB Inputs/Value Channel 14 <-> Data Pointer/RawPositionValues[13]
//     Term 11 (AT2050-0500)/Term 12 (AT2050-5500)/FB Inputs/Value Channel 15 <-> Data Pointer/RawPositionValues[14]
//     Term 11 (AT2050-0500)/Term 12 (AT2050-5500)/FB Inputs/Value Channel 16 <-> Data Pointer/RawPositionValues[15]
//     Term 11 (AT2050-0500)/Term 12 (AT2050-5500)/FB Inputs/Value Channel 17 <-> Data Pointer/RawPositionValues[16]
//     Term 11 (AT2050-0500)/Term 12 (AT2050-5500)/FB Inputs/Value Channel 18 <-> Data Pointer/RawPositionValues[17]
//     Term 11 (AT2050-0500)/Term 12 (AT2050-5500)/FB Inputs/Value Channel 19 <-> Data Pointer/RawPositionValues[18]
//     Term 11 (AT2050-0500)/Term 12 (AT2050-5500)/FB Inputs/Value Channel 20 <-> Data Pointer/RawPositionValues[19]
//     Term 11 (AT2050-0500)/Term 12 (AT2050-5500)/FB Inputs/Value Channel 21 <-> Data Pointer/RawPositionValues[20]
//     Term 11 (AT2050-0500)/Term 12 (AT2050-5500)/FB Inputs/Value Channel 22 <-> Data Pointer/RawPositionValues[21]
//     Term 11 (AT2050-0500)/Term 12 (AT2050-5500)/FB Inputs/Value Channel 23 <-> Data Pointer/RawPositionValues[22]
//     Term 11 (AT2050-0500)/Term 12 (AT2050-5500)/FB Inputs/Value Channel 24 <-> Data Pointer/RawPositionValues[23]
//     Term 11 (AT2050-0500)/Term 12 (AT2050-5500)/FB Inputs/Value Channel 25 <-> Data Pointer/RawPositionValues[24]
//     Term 11 (AT2050-0500)/Term 12 (AT2050-5500)/FB Inputs/Value Channel 26 <-> Data Pointer/RawPositionValues[25]
//     Term 11 (AT2050-0500)/Term 12 (AT2050-5500)/FB Inputs/Value Channel 27 <-> Data Pointer/RawPositionValues[26]
//     Term 11 (AT2050-0500)/Term 12 (AT2050-5500)/FB Inputs/Value Channel 28 <-> Data Pointer/RawPositionValues[27]
//     Term 11 (AT2050-0500)/Term 12 (AT2050-5500)/FB Inputs/Value Channel 29 <-> Data Pointer/RawPositionValues[28]
//     Term 11 (AT2050-0500)/Term 12 (AT2050-5500)/FB Inputs/Value Channel 30 <-> Data Pointer/RawPositionValues[29]
//     Term 11 (AT2050-0500)/Term 12 (AT2050-5500)/FB Inputs/Value Channel 31 <-> Data Pointer/RawPositionValues[30]
//     Term 11 (AT2050-0500)/Term 12 (AT2050-5500)/FB Inputs/Value Channel 32 <-> Data Pointer/RawPositionValues[31]
//   Device 6 (EtherCAT) <-> TcCOM Objects/XtsProcessingUnit 1/Part 1/Module 6
//     Term 13 (AT2050-0501)/CC Inputs/Current actual value Ch.1 <-> Data Pointer/CurrentActualValues[0]
//     Term 13 (AT2050-0501)/CC Inputs/Current actual value Ch.10 <-> Data Pointer/CurrentActualValues[9]
//     Term 13 (AT2050-0501)/CC Inputs/Current actual value Ch.11 <-> Data Pointer/CurrentActualValues[10]
//     Term 13 (AT2050-0501)/CC Inputs/Current actual value Ch.12 <-> Data Pointer/CurrentActualValues[11]
//     Term 13 (AT2050-0501)/CC Inputs/Current actual value Ch.13 <-> Data Pointer/CurrentActualValues[12]
//     Term 13 (AT2050-0501)/CC Inputs/Current actual value Ch.14 <-> Data Pointer/CurrentActualValues[13]
//     Term 13 (AT2050-0501)/CC Inputs/Current actual value Ch.15 <-> Data Pointer/CurrentActualValues[14]
//     Term 13 (AT2050-0501)/CC Inputs/Current actual value Ch.2 <-> Data Pointer/CurrentActualValues[1]
//     Term 13 (AT2050-0501)/CC Inputs/Current actual value Ch.3 <-> Data Pointer/CurrentActualValues[2]
//     Term 13 (AT2050-0501)/CC Inputs/Current actual value Ch.4 <-> Data Pointer/CurrentActualValues[3]
//     Term 13 (AT2050-0501)/CC Inputs/Current actual value Ch.5 <-> Data Pointer/CurrentActualValues[4]
//     Term 13 (AT2050-0501)/CC Inputs/Current actual value Ch.6 <-> Data Pointer/CurrentActualValues[5]
//     Term 13 (AT2050-0501)/CC Inputs/Current actual value Ch.7 <-> Data Pointer/CurrentActualValues[6]
//     Term 13 (AT2050-0501)/CC Inputs/Current actual value Ch.8 <-> Data Pointer/CurrentActualValues[7]
//     Term 13 (AT2050-0501)/CC Inputs/Current actual value Ch.9 <-> Data Pointer/CurrentActualValues[8]
//     Term 13 (AT2050-0501)/CC Inputs/Status <-> Data Pointer/Status
//     Term 13 (AT2050-0501)/CC Outputs/Control <-> Data Pointer/Control
//     Term 13 (AT2050-0501)/CC Outputs/Current setpoint value Ch.1 <-> Data Pointer/CurrentSetpointValues[0]
//     Term 13 (AT2050-0501)/CC Outputs/Current setpoint value Ch.10 <-> Data Pointer/CurrentSetpointValues[9]
//     Term 13 (AT2050-0501)/CC Outputs/Current setpoint value Ch.11 <-> Data Pointer/CurrentSetpointValues[10]
//     Term 13 (AT2050-0501)/CC Outputs/Current setpoint value Ch.12 <-> Data Pointer/CurrentSetpointValues[11]
//     Term 13 (AT2050-0501)/CC Outputs/Current setpoint value Ch.13 <-> Data Pointer/CurrentSetpointValues[12]
//     Term 13 (AT2050-0501)/CC Outputs/Current setpoint value Ch.14 <-> Data Pointer/CurrentSetpointValues[13]
//     Term 13 (AT2050-0501)/CC Outputs/Current setpoint value Ch.15 <-> Data Pointer/CurrentSetpointValues[14]
//     Term 13 (AT2050-0501)/CC Outputs/Current setpoint value Ch.2 <-> Data Pointer/CurrentSetpointValues[1]
//     Term 13 (AT2050-0501)/CC Outputs/Current setpoint value Ch.3 <-> Data Pointer/CurrentSetpointValues[2]
//     Term 13 (AT2050-0501)/CC Outputs/Current setpoint value Ch.4 <-> Data Pointer/CurrentSetpointValues[3]
//     Term 13 (AT2050-0501)/CC Outputs/Current setpoint value Ch.5 <-> Data Pointer/CurrentSetpointValues[4]
//     Term 13 (AT2050-0501)/CC Outputs/Current setpoint value Ch.6 <-> Data Pointer/CurrentSetpointValues[5]
//     Term 13 (AT2050-0501)/CC Outputs/Current setpoint value Ch.7 <-> Data Pointer/CurrentSetpointValues[6]
//     Term 13 (AT2050-0501)/CC Outputs/Current setpoint value Ch.8 <-> Data Pointer/CurrentSetpointValues[7]
//     Term 13 (AT2050-0501)/CC Outputs/Current setpoint value Ch.9 <-> Data Pointer/CurrentSetpointValues[8]
//     Term 13 (AT2050-0501)/Term 14 (AT2050-5501)/FB Inputs/Value Channel 01 <-> Data Pointer/RawPositionValues[0]
//     Term 13 (AT2050-0501)/Term 14 (AT2050-5501)/FB Inputs/Value Channel 02 <-> Data Pointer/RawPositionValues[1]
//     Term 13 (AT2050-0501)/Term 14 (AT2050-5501)/FB Inputs/Value Channel 03 <-> Data Pointer/RawPositionValues[2]
//     Term 13 (AT2050-0501)/Term 14 (AT2050-5501)/FB Inputs/Value Channel 04 <-> Data Pointer/RawPositionValues[3]
//     Term 13 (AT2050-0501)/Term 14 (AT2050-5501)/FB Inputs/Value Channel 05 <-> Data Pointer/RawPositionValues[4]
//     Term 13 (AT2050-0501)/Term 14 (AT2050-5501)/FB Inputs/Value Channel 06 <-> Data Pointer/RawPositionValues[5]
//     Term 13 (AT2050-0501)/Term 14 (AT2050-5501)/FB Inputs/Value Channel 07 <-> Data Pointer/RawPositionValues[6]
//     Term 13 (AT2050-0501)/Term 14 (AT2050-5501)/FB Inputs/Value Channel 08 <-> Data Pointer/RawPositionValues[7]
//     Term 13 (AT2050-0501)/Term 14 (AT2050-5501)/FB Inputs/Value Channel 09 <-> Data Pointer/RawPositionValues[8]
//     Term 13 (AT2050-0501)/Term 14 (AT2050-5501)/FB Inputs/Value Channel 10 <-> Data Pointer/RawPositionValues[9]
//     Term 13 (AT2050-0501)/Term 14 (AT2050-5501)/FB Inputs/Value Channel 11 <-> Data Pointer/RawPositionValues[10]
//     Term 13 (AT2050-0501)/Term 14 (AT2050-5501)/FB Inputs/Value Channel 12 <-> Data Pointer/RawPositionValues[11]
//     Term 13 (AT2050-0501)/Term 14 (AT2050-5501)/FB Inputs/Value Channel 13 <-> Data Pointer/RawPositionValues[12]
//     Term 13 (AT2050-0501)/Term 14 (AT2050-5501)/FB Inputs/Value Channel 14 <-> Data Pointer/RawPositionValues[13]
//     Term 13 (AT2050-0501)/Term 14 (AT2050-5501)/FB Inputs/Value Channel 15 <-> Data Pointer/RawPositionValues[14]
//     Term 13 (AT2050-0501)/Term 14 (AT2050-5501)/FB Inputs/Value Channel 16 <-> Data Pointer/RawPositionValues[15]
//     Term 13 (AT2050-0501)/Term 14 (AT2050-5501)/FB Inputs/Value Channel 17 <-> Data Pointer/RawPositionValues[16]
//     Term 13 (AT2050-0501)/Term 14 (AT2050-5501)/FB Inputs/Value Channel 18 <-> Data Pointer/RawPositionValues[17]
//     Term 13 (AT2050-0501)/Term 14 (AT2050-5501)/FB Inputs/Value Channel 19 <-> Data Pointer/RawPositionValues[18]
//     Term 13 (AT2050-0501)/Term 14 (AT2050-5501)/FB Inputs/Value Channel 20 <-> Data Pointer/RawPositionValues[19]
//     Term 13 (AT2050-0501)/Term 14 (AT2050-5501)/FB Inputs/Value Channel 21 <-> Data Pointer/RawPositionValues[20]
//     Term 13 (AT2050-0501)/Term 14 (AT2050-5501)/FB Inputs/Value Channel 22 <-> Data Pointer/RawPositionValues[21]
//     Term 13 (AT2050-0501)/Term 14 (AT2050-5501)/FB Inputs/Value Channel 23 <-> Data Pointer/RawPositionValues[22]
//     Term 13 (AT2050-0501)/Term 14 (AT2050-5501)/FB Inputs/Value Channel 24 <-> Data Pointer/RawPositionValues[23]
//     Term 13 (AT2050-0501)/Term 14 (AT2050-5501)/FB Inputs/Value Channel 25 <-> Data Pointer/RawPositionValues[24]
//     Term 13 (AT2050-0501)/Term 14 (AT2050-5501)/FB Inputs/Value Channel 26 <-> Data Pointer/RawPositionValues[25]
//     Term 13 (AT2050-0501)/Term 14 (AT2050-5501)/FB Inputs/Value Channel 27 <-> Data Pointer/RawPositionValues[26]
//     Term 13 (AT2050-0501)/Term 14 (AT2050-5501)/FB Inputs/Value Channel 28 <-> Data Pointer/RawPositionValues[27]
//     Term 13 (AT2050-0501)/Term 14 (AT2050-5501)/FB Inputs/Value Channel 29 <-> Data Pointer/RawPositionValues[28]
//     Term 13 (AT2050-0501)/Term 14 (AT2050-5501)/FB Inputs/Value Channel 30 <-> Data Pointer/RawPositionValues[29]
//     Term 13 (AT2050-0501)/Term 14 (AT2050-5501)/FB Inputs/Value Channel 31 <-> Data Pointer/RawPositionValues[30]
//     Term 13 (AT2050-0501)/Term 14 (AT2050-5501)/FB Inputs/Value Channel 32 <-> Data Pointer/RawPositionValues[31]
//   Device 7 (EtherCAT) <-> TcCOM Objects/XtsProcessingUnit 1/Part 1/Module 7
//     Term 16 (AT2001-0250)/CC Inputs/Current actual value Ch.1 <-> Data Pointer/CurrentActualValues[0]
//     Term 16 (AT2001-0250)/CC Inputs/Current actual value Ch.10 <-> Data Pointer/CurrentActualValues[9]
//     Term 16 (AT2001-0250)/CC Inputs/Current actual value Ch.11 <-> Data Pointer/CurrentActualValues[10]
//     Term 16 (AT2001-0250)/CC Inputs/Current actual value Ch.12 <-> Data Pointer/CurrentActualValues[11]
//     Term 16 (AT2001-0250)/CC Inputs/Current actual value Ch.13 <-> Data Pointer/CurrentActualValues[12]
//     Term 16 (AT2001-0250)/CC Inputs/Current actual value Ch.14 <-> Data Pointer/CurrentActualValues[13]
//     Term 16 (AT2001-0250)/CC Inputs/Current actual value Ch.15 <-> Data Pointer/CurrentActualValues[14]
//     Term 16 (AT2001-0250)/CC Inputs/Current actual value Ch.2 <-> Data Pointer/CurrentActualValues[1]
//     Term 16 (AT2001-0250)/CC Inputs/Current actual value Ch.3 <-> Data Pointer/CurrentActualValues[2]
//     Term 16 (AT2001-0250)/CC Inputs/Current actual value Ch.4 <-> Data Pointer/CurrentActualValues[3]
//     Term 16 (AT2001-0250)/CC Inputs/Current actual value Ch.5 <-> Data Pointer/CurrentActualValues[4]
//     Term 16 (AT2001-0250)/CC Inputs/Current actual value Ch.6 <-> Data Pointer/CurrentActualValues[5]
//     Term 16 (AT2001-0250)/CC Inputs/Current actual value Ch.7 <-> Data Pointer/CurrentActualValues[6]
//     Term 16 (AT2001-0250)/CC Inputs/Current actual value Ch.8 <-> Data Pointer/CurrentActualValues[7]
//     Term 16 (AT2001-0250)/CC Inputs/Current actual value Ch.9 <-> Data Pointer/CurrentActualValues[8]
//     Term 16 (AT2001-0250)/CC Inputs/Status <-> Data Pointer/Status
//     Term 16 (AT2001-0250)/CC Outputs/Control <-> Data Pointer/Control
//     Term 16 (AT2001-0250)/CC Outputs/Current setpoint value Ch.1 <-> Data Pointer/CurrentSetpointValues[0]
//     Term 16 (AT2001-0250)/CC Outputs/Current setpoint value Ch.10 <-> Data Pointer/CurrentSetpointValues[9]
//     Term 16 (AT2001-0250)/CC Outputs/Current setpoint value Ch.11 <-> Data Pointer/CurrentSetpointValues[10]
//     Term 16 (AT2001-0250)/CC Outputs/Current setpoint value Ch.12 <-> Data Pointer/CurrentSetpointValues[11]
//     Term 16 (AT2001-0250)/CC Outputs/Current setpoint value Ch.13 <-> Data Pointer/CurrentSetpointValues[12]
//     Term 16 (AT2001-0250)/CC Outputs/Current setpoint value Ch.14 <-> Data Pointer/CurrentSetpointValues[13]
//     Term 16 (AT2001-0250)/CC Outputs/Current setpoint value Ch.15 <-> Data Pointer/CurrentSetpointValues[14]
//     Term 16 (AT2001-0250)/CC Outputs/Current setpoint value Ch.2 <-> Data Pointer/CurrentSetpointValues[1]
//     Term 16 (AT2001-0250)/CC Outputs/Current setpoint value Ch.3 <-> Data Pointer/CurrentSetpointValues[2]
//     Term 16 (AT2001-0250)/CC Outputs/Current setpoint value Ch.4 <-> Data Pointer/CurrentSetpointValues[3]
//     Term 16 (AT2001-0250)/CC Outputs/Current setpoint value Ch.5 <-> Data Pointer/CurrentSetpointValues[4]
//     Term 16 (AT2001-0250)/CC Outputs/Current setpoint value Ch.6 <-> Data Pointer/CurrentSetpointValues[5]
//     Term 16 (AT2001-0250)/CC Outputs/Current setpoint value Ch.7 <-> Data Pointer/CurrentSetpointValues[6]
//     Term 16 (AT2001-0250)/CC Outputs/Current setpoint value Ch.8 <-> Data Pointer/CurrentSetpointValues[7]
//     Term 16 (AT2001-0250)/CC Outputs/Current setpoint value Ch.9 <-> Data Pointer/CurrentSetpointValues[8]
//     Term 16 (AT2001-0250)/Term 17 (AT2001-5250)/FB Inputs/Value Channel 01 <-> Data Pointer/RawPositionValues[0]
//     Term 16 (AT2001-0250)/Term 17 (AT2001-5250)/FB Inputs/Value Channel 02 <-> Data Pointer/RawPositionValues[1]
//     Term 16 (AT2001-0250)/Term 17 (AT2001-5250)/FB Inputs/Value Channel 03 <-> Data Pointer/RawPositionValues[2]
//     Term 16 (AT2001-0250)/Term 17 (AT2001-5250)/FB Inputs/Value Channel 04 <-> Data Pointer/RawPositionValues[3]
//     Term 16 (AT2001-0250)/Term 17 (AT2001-5250)/FB Inputs/Value Channel 05 <-> Data Pointer/RawPositionValues[4]
//     Term 16 (AT2001-0250)/Term 17 (AT2001-5250)/FB Inputs/Value Channel 06 <-> Data Pointer/RawPositionValues[5]
//     Term 16 (AT2001-0250)/Term 17 (AT2001-5250)/FB Inputs/Value Channel 07 <-> Data Pointer/RawPositionValues[6]
//     Term 16 (AT2001-0250)/Term 17 (AT2001-5250)/FB Inputs/Value Channel 08 <-> Data Pointer/RawPositionValues[7]
//     Term 16 (AT2001-0250)/Term 17 (AT2001-5250)/FB Inputs/Value Channel 09 <-> Data Pointer/RawPositionValues[8]
//     Term 16 (AT2001-0250)/Term 17 (AT2001-5250)/FB Inputs/Value Channel 10 <-> Data Pointer/RawPositionValues[9]
//     Term 16 (AT2001-0250)/Term 17 (AT2001-5250)/FB Inputs/Value Channel 11 <-> Data Pointer/RawPositionValues[10]
//     Term 16 (AT2001-0250)/Term 17 (AT2001-5250)/FB Inputs/Value Channel 12 <-> Data Pointer/RawPositionValues[11]
//     Term 16 (AT2001-0250)/Term 17 (AT2001-5250)/FB Inputs/Value Channel 13 <-> Data Pointer/RawPositionValues[12]
//     Term 16 (AT2001-0250)/Term 17 (AT2001-5250)/FB Inputs/Value Channel 14 <-> Data Pointer/RawPositionValues[13]
//     Term 16 (AT2001-0250)/Term 17 (AT2001-5250)/FB Inputs/Value Channel 15 <-> Data Pointer/RawPositionValues[14]
//     Term 16 (AT2001-0250)/Term 17 (AT2001-5250)/FB Inputs/Value Channel 16 <-> Data Pointer/RawPositionValues[15]
//     Term 16 (AT2001-0250)/Term 17 (AT2001-5250)/FB Inputs/Value Channel 17 <-> Data Pointer/RawPositionValues[16]
//     Term 16 (AT2001-0250)/Term 17 (AT2001-5250)/FB Inputs/Value Channel 18 <-> Data Pointer/RawPositionValues[17]
//     Term 16 (AT2001-0250)/Term 17 (AT2001-5250)/FB Inputs/Value Channel 19 <-> Data Pointer/RawPositionValues[18]
//     Term 16 (AT2001-0250)/Term 17 (AT2001-5250)/FB Inputs/Value Channel 20 <-> Data Pointer/RawPositionValues[19]
//     Term 16 (AT2001-0250)/Term 17 (AT2001-5250)/FB Inputs/Value Channel 21 <-> Data Pointer/RawPositionValues[20]
//     Term 16 (AT2001-0250)/Term 17 (AT2001-5250)/FB Inputs/Value Channel 22 <-> Data Pointer/RawPositionValues[21]
//     Term 16 (AT2001-0250)/Term 17 (AT2001-5250)/FB Inputs/Value Channel 23 <-> Data Pointer/RawPositionValues[22]
//     Term 16 (AT2001-0250)/Term 17 (AT2001-5250)/FB Inputs/Value Channel 24 <-> Data Pointer/RawPositionValues[23]
//     Term 16 (AT2001-0250)/Term 17 (AT2001-5250)/FB Inputs/Value Channel 25 <-> Data Pointer/RawPositionValues[24]
//     Term 16 (AT2001-0250)/Term 17 (AT2001-5250)/FB Inputs/Value Channel 26 <-> Data Pointer/RawPositionValues[25]
//     Term 16 (AT2001-0250)/Term 17 (AT2001-5250)/FB Inputs/Value Channel 27 <-> Data Pointer/RawPositionValues[26]
//     Term 16 (AT2001-0250)/Term 17 (AT2001-5250)/FB Inputs/Value Channel 28 <-> Data Pointer/RawPositionValues[27]
//     Term 16 (AT2001-0250)/Term 17 (AT2001-5250)/FB Inputs/Value Channel 29 <-> Data Pointer/RawPositionValues[28]
//     Term 16 (AT2001-0250)/Term 17 (AT2001-5250)/FB Inputs/Value Channel 30 <-> Data Pointer/RawPositionValues[29]
//     Term 16 (AT2001-0250)/Term 17 (AT2001-5250)/FB Inputs/Value Channel 31 <-> Data Pointer/RawPositionValues[30]
//     Term 16 (AT2001-0250)/Term 17 (AT2001-5250)/FB Inputs/Value Channel 32 <-> Data Pointer/RawPositionValues[31]
//   Device 7 (EtherCAT) <-> TcCOM Objects/XtsProcessingUnit 1/Part 1/Module 8
//     Term 18 (AT2000-0250)/CC Inputs/Current actual value Ch.1 <-> Data Pointer/CurrentActualValues[0]
//     Term 18 (AT2000-0250)/CC Inputs/Current actual value Ch.10 <-> Data Pointer/CurrentActualValues[9]
//     Term 18 (AT2000-0250)/CC Inputs/Current actual value Ch.11 <-> Data Pointer/CurrentActualValues[10]
//     Term 18 (AT2000-0250)/CC Inputs/Current actual value Ch.12 <-> Data Pointer/CurrentActualValues[11]
//     Term 18 (AT2000-0250)/CC Inputs/Current actual value Ch.13 <-> Data Pointer/CurrentActualValues[12]
//     Term 18 (AT2000-0250)/CC Inputs/Current actual value Ch.14 <-> Data Pointer/CurrentActualValues[13]
//     Term 18 (AT2000-0250)/CC Inputs/Current actual value Ch.15 <-> Data Pointer/CurrentActualValues[14]
//     Term 18 (AT2000-0250)/CC Inputs/Current actual value Ch.2 <-> Data Pointer/CurrentActualValues[1]
//     Term 18 (AT2000-0250)/CC Inputs/Current actual value Ch.3 <-> Data Pointer/CurrentActualValues[2]
//     Term 18 (AT2000-0250)/CC Inputs/Current actual value Ch.4 <-> Data Pointer/CurrentActualValues[3]
//     Term 18 (AT2000-0250)/CC Inputs/Current actual value Ch.5 <-> Data Pointer/CurrentActualValues[4]
//     Term 18 (AT2000-0250)/CC Inputs/Current actual value Ch.6 <-> Data Pointer/CurrentActualValues[5]
//     Term 18 (AT2000-0250)/CC Inputs/Current actual value Ch.7 <-> Data Pointer/CurrentActualValues[6]
//     Term 18 (AT2000-0250)/CC Inputs/Current actual value Ch.8 <-> Data Pointer/CurrentActualValues[7]
//     Term 18 (AT2000-0250)/CC Inputs/Current actual value Ch.9 <-> Data Pointer/CurrentActualValues[8]
//     Term 18 (AT2000-0250)/CC Inputs/Status <-> Data Pointer/Status
//     Term 18 (AT2000-0250)/CC Outputs/Control <-> Data Pointer/Control
//     Term 18 (AT2000-0250)/CC Outputs/Current setpoint value Ch.1 <-> Data Pointer/CurrentSetpointValues[0]
//     Term 18 (AT2000-0250)/CC Outputs/Current setpoint value Ch.10 <-> Data Pointer/CurrentSetpointValues[9]
//     Term 18 (AT2000-0250)/CC Outputs/Current setpoint value Ch.11 <-> Data Pointer/CurrentSetpointValues[10]
//     Term 18 (AT2000-0250)/CC Outputs/Current setpoint value Ch.12 <-> Data Pointer/CurrentSetpointValues[11]
//     Term 18 (AT2000-0250)/CC Outputs/Current setpoint value Ch.13 <-> Data Pointer/CurrentSetpointValues[12]
//     Term 18 (AT2000-0250)/CC Outputs/Current setpoint value Ch.14 <-> Data Pointer/CurrentSetpointValues[13]
//     Term 18 (AT2000-0250)/CC Outputs/Current setpoint value Ch.15 <-> Data Pointer/CurrentSetpointValues[14]
//     Term 18 (AT2000-0250)/CC Outputs/Current setpoint value Ch.2 <-> Data Pointer/CurrentSetpointValues[1]
//     Term 18 (AT2000-0250)/CC Outputs/Current setpoint value Ch.3 <-> Data Pointer/CurrentSetpointValues[2]
//     Term 18 (AT2000-0250)/CC Outputs/Current setpoint value Ch.4 <-> Data Pointer/CurrentSetpointValues[3]
//     Term 18 (AT2000-0250)/CC Outputs/Current setpoint value Ch.5 <-> Data Pointer/CurrentSetpointValues[4]
//     Term 18 (AT2000-0250)/CC Outputs/Current setpoint value Ch.6 <-> Data Pointer/CurrentSetpointValues[5]
//     Term 18 (AT2000-0250)/CC Outputs/Current setpoint value Ch.7 <-> Data Pointer/CurrentSetpointValues[6]
//     Term 18 (AT2000-0250)/CC Outputs/Current setpoint value Ch.8 <-> Data Pointer/CurrentSetpointValues[7]
//     Term 18 (AT2000-0250)/CC Outputs/Current setpoint value Ch.9 <-> Data Pointer/CurrentSetpointValues[8]
//     Term 18 (AT2000-0250)/Term 19 (AT2000-5250)/FB Inputs/Value Channel 01 <-> Data Pointer/RawPositionValues[0]
//     Term 18 (AT2000-0250)/Term 19 (AT2000-5250)/FB Inputs/Value Channel 02 <-> Data Pointer/RawPositionValues[1]
//     Term 18 (AT2000-0250)/Term 19 (AT2000-5250)/FB Inputs/Value Channel 03 <-> Data Pointer/RawPositionValues[2]
//     Term 18 (AT2000-0250)/Term 19 (AT2000-5250)/FB Inputs/Value Channel 04 <-> Data Pointer/RawPositionValues[3]
//     Term 18 (AT2000-0250)/Term 19 (AT2000-5250)/FB Inputs/Value Channel 05 <-> Data Pointer/RawPositionValues[4]
//     Term 18 (AT2000-0250)/Term 19 (AT2000-5250)/FB Inputs/Value Channel 06 <-> Data Pointer/RawPositionValues[5]
//     Term 18 (AT2000-0250)/Term 19 (AT2000-5250)/FB Inputs/Value Channel 07 <-> Data Pointer/RawPositionValues[6]
//     Term 18 (AT2000-0250)/Term 19 (AT2000-5250)/FB Inputs/Value Channel 08 <-> Data Pointer/RawPositionValues[7]
//     Term 18 (AT2000-0250)/Term 19 (AT2000-5250)/FB Inputs/Value Channel 09 <-> Data Pointer/RawPositionValues[8]
//     Term 18 (AT2000-0250)/Term 19 (AT2000-5250)/FB Inputs/Value Channel 10 <-> Data Pointer/RawPositionValues[9]
//     Term 18 (AT2000-0250)/Term 19 (AT2000-5250)/FB Inputs/Value Channel 11 <-> Data Pointer/RawPositionValues[10]
//     Term 18 (AT2000-0250)/Term 19 (AT2000-5250)/FB Inputs/Value Channel 12 <-> Data Pointer/RawPositionValues[11]
//     Term 18 (AT2000-0250)/Term 19 (AT2000-5250)/FB Inputs/Value Channel 13 <-> Data Pointer/RawPositionValues[12]
//     Term 18 (AT2000-0250)/Term 19 (AT2000-5250)/FB Inputs/Value Channel 14 <-> Data Pointer/RawPositionValues[13]
//     Term 18 (AT2000-0250)/Term 19 (AT2000-5250)/FB Inputs/Value Channel 15 <-> Data Pointer/RawPositionValues[14]
//     Term 18 (AT2000-0250)/Term 19 (AT2000-5250)/FB Inputs/Value Channel 16 <-> Data Pointer/RawPositionValues[15]
//     Term 18 (AT2000-0250)/Term 19 (AT2000-5250)/FB Inputs/Value Channel 17 <-> Data Pointer/RawPositionValues[16]
//     Term 18 (AT2000-0250)/Term 19 (AT2000-5250)/FB Inputs/Value Channel 18 <-> Data Pointer/RawPositionValues[17]
//     Term 18 (AT2000-0250)/Term 19 (AT2000-5250)/FB Inputs/Value Channel 19 <-> Data Pointer/RawPositionValues[18]
//     Term 18 (AT2000-0250)/Term 19 (AT2000-5250)/FB Inputs/Value Channel 20 <-> Data Pointer/RawPositionValues[19]
//     Term 18 (AT2000-0250)/Term 19 (AT2000-5250)/FB Inputs/Value Channel 21 <-> Data Pointer/RawPositionValues[20]
//     Term 18 (AT2000-0250)/Term 19 (AT2000-5250)/FB Inputs/Value Channel 22 <-> Data Pointer/RawPositionValues[21]
//     Term 18 (AT2000-0250)/Term 19 (AT2000-5250)/FB Inputs/Value Channel 23 <-> Data Pointer/RawPositionValues[22]
//     Term 18 (AT2000-0250)/Term 19 (AT2000-5250)/FB Inputs/Value Channel 24 <-> Data Pointer/RawPositionValues[23]
//     Term 18 (AT2000-0250)/Term 19 (AT2000-5250)/FB Inputs/Value Channel 25 <-> Data Pointer/RawPositionValues[24]
//     Term 18 (AT2000-0250)/Term 19 (AT2000-5250)/FB Inputs/Value Channel 26 <-> Data Pointer/RawPositionValues[25]
//     Term 18 (AT2000-0250)/Term 19 (AT2000-5250)/FB Inputs/Value Channel 27 <-> Data Pointer/RawPositionValues[26]
//     Term 18 (AT2000-0250)/Term 19 (AT2000-5250)/FB Inputs/Value Channel 28 <-> Data Pointer/RawPositionValues[27]
//     Term 18 (AT2000-0250)/Term 19 (AT2000-5250)/FB Inputs/Value Channel 29 <-> Data Pointer/RawPositionValues[28]
//     Term 18 (AT2000-0250)/Term 19 (AT2000-5250)/FB Inputs/Value Channel 30 <-> Data Pointer/RawPositionValues[29]
//     Term 18 (AT2000-0250)/Term 19 (AT2000-5250)/FB Inputs/Value Channel 31 <-> Data Pointer/RawPositionValues[30]
//     Term 18 (AT2000-0250)/Term 19 (AT2000-5250)/FB Inputs/Value Channel 32 <-> Data Pointer/RawPositionValues[31]
//   Device 7 (EtherCAT) <-> TcCOM Objects/XtsProcessingUnit 1/Part 1/Module 9
//     Term 20 (AT2000-0250)/CC Inputs/Current actual value Ch.1 <-> Data Pointer/CurrentActualValues[0]
//     Term 20 (AT2000-0250)/CC Inputs/Current actual value Ch.10 <-> Data Pointer/CurrentActualValues[9]
//     Term 20 (AT2000-0250)/CC Inputs/Current actual value Ch.11 <-> Data Pointer/CurrentActualValues[10]
//     Term 20 (AT2000-0250)/CC Inputs/Current actual value Ch.12 <-> Data Pointer/CurrentActualValues[11]
//     Term 20 (AT2000-0250)/CC Inputs/Current actual value Ch.13 <-> Data Pointer/CurrentActualValues[12]
//     Term 20 (AT2000-0250)/CC Inputs/Current actual value Ch.14 <-> Data Pointer/CurrentActualValues[13]
//     Term 20 (AT2000-0250)/CC Inputs/Current actual value Ch.15 <-> Data Pointer/CurrentActualValues[14]
//     Term 20 (AT2000-0250)/CC Inputs/Current actual value Ch.2 <-> Data Pointer/CurrentActualValues[1]
//     Term 20 (AT2000-0250)/CC Inputs/Current actual value Ch.3 <-> Data Pointer/CurrentActualValues[2]
//     Term 20 (AT2000-0250)/CC Inputs/Current actual value Ch.4 <-> Data Pointer/CurrentActualValues[3]
//     Term 20 (AT2000-0250)/CC Inputs/Current actual value Ch.5 <-> Data Pointer/CurrentActualValues[4]
//     Term 20 (AT2000-0250)/CC Inputs/Current actual value Ch.6 <-> Data Pointer/CurrentActualValues[5]
//     Term 20 (AT2000-0250)/CC Inputs/Current actual value Ch.7 <-> Data Pointer/CurrentActualValues[6]
//     Term 20 (AT2000-0250)/CC Inputs/Current actual value Ch.8 <-> Data Pointer/CurrentActualValues[7]
//     Term 20 (AT2000-0250)/CC Inputs/Current actual value Ch.9 <-> Data Pointer/CurrentActualValues[8]
//     Term 20 (AT2000-0250)/CC Inputs/Status <-> Data Pointer/Status
//     Term 20 (AT2000-0250)/CC Outputs/Control <-> Data Pointer/Control
//     Term 20 (AT2000-0250)/CC Outputs/Current setpoint value Ch.1 <-> Data Pointer/CurrentSetpointValues[0]
//     Term 20 (AT2000-0250)/CC Outputs/Current setpoint value Ch.10 <-> Data Pointer/CurrentSetpointValues[9]
//     Term 20 (AT2000-0250)/CC Outputs/Current setpoint value Ch.11 <-> Data Pointer/CurrentSetpointValues[10]
//     Term 20 (AT2000-0250)/CC Outputs/Current setpoint value Ch.12 <-> Data Pointer/CurrentSetpointValues[11]
//     Term 20 (AT2000-0250)/CC Outputs/Current setpoint value Ch.13 <-> Data Pointer/CurrentSetpointValues[12]
//     Term 20 (AT2000-0250)/CC Outputs/Current setpoint value Ch.14 <-> Data Pointer/CurrentSetpointValues[13]
//     Term 20 (AT2000-0250)/CC Outputs/Current setpoint value Ch.15 <-> Data Pointer/CurrentSetpointValues[14]
//     Term 20 (AT2000-0250)/CC Outputs/Current setpoint value Ch.2 <-> Data Pointer/CurrentSetpointValues[1]
//     Term 20 (AT2000-0250)/CC Outputs/Current setpoint value Ch.3 <-> Data Pointer/CurrentSetpointValues[2]
//     Term 20 (AT2000-0250)/CC Outputs/Current setpoint value Ch.4 <-> Data Pointer/CurrentSetpointValues[3]
//     Term 20 (AT2000-0250)/CC Outputs/Current setpoint value Ch.5 <-> Data Pointer/CurrentSetpointValues[4]
//     Term 20 (AT2000-0250)/CC Outputs/Current setpoint value Ch.6 <-> Data Pointer/CurrentSetpointValues[5]
//     Term 20 (AT2000-0250)/CC Outputs/Current setpoint value Ch.7 <-> Data Pointer/CurrentSetpointValues[6]
//     Term 20 (AT2000-0250)/CC Outputs/Current setpoint value Ch.8 <-> Data Pointer/CurrentSetpointValues[7]
//     Term 20 (AT2000-0250)/CC Outputs/Current setpoint value Ch.9 <-> Data Pointer/CurrentSetpointValues[8]
//     Term 20 (AT2000-0250)/Term 21 (AT2000-5250)/FB Inputs/Value Channel 01 <-> Data Pointer/RawPositionValues[0]
//     Term 20 (AT2000-0250)/Term 21 (AT2000-5250)/FB Inputs/Value Channel 02 <-> Data Pointer/RawPositionValues[1]
//     Term 20 (AT2000-0250)/Term 21 (AT2000-5250)/FB Inputs/Value Channel 03 <-> Data Pointer/RawPositionValues[2]
//     Term 20 (AT2000-0250)/Term 21 (AT2000-5250)/FB Inputs/Value Channel 04 <-> Data Pointer/RawPositionValues[3]
//     Term 20 (AT2000-0250)/Term 21 (AT2000-5250)/FB Inputs/Value Channel 05 <-> Data Pointer/RawPositionValues[4]
//     Term 20 (AT2000-0250)/Term 21 (AT2000-5250)/FB Inputs/Value Channel 06 <-> Data Pointer/RawPositionValues[5]
//     Term 20 (AT2000-0250)/Term 21 (AT2000-5250)/FB Inputs/Value Channel 07 <-> Data Pointer/RawPositionValues[6]
//     Term 20 (AT2000-0250)/Term 21 (AT2000-5250)/FB Inputs/Value Channel 08 <-> Data Pointer/RawPositionValues[7]
//     Term 20 (AT2000-0250)/Term 21 (AT2000-5250)/FB Inputs/Value Channel 09 <-> Data Pointer/RawPositionValues[8]
//     Term 20 (AT2000-0250)/Term 21 (AT2000-5250)/FB Inputs/Value Channel 10 <-> Data Pointer/RawPositionValues[9]
//     Term 20 (AT2000-0250)/Term 21 (AT2000-5250)/FB Inputs/Value Channel 11 <-> Data Pointer/RawPositionValues[10]
//     Term 20 (AT2000-0250)/Term 21 (AT2000-5250)/FB Inputs/Value Channel 12 <-> Data Pointer/RawPositionValues[11]
//     Term 20 (AT2000-0250)/Term 21 (AT2000-5250)/FB Inputs/Value Channel 13 <-> Data Pointer/RawPositionValues[12]
//     Term 20 (AT2000-0250)/Term 21 (AT2000-5250)/FB Inputs/Value Channel 14 <-> Data Pointer/RawPositionValues[13]
//     Term 20 (AT2000-0250)/Term 21 (AT2000-5250)/FB Inputs/Value Channel 15 <-> Data Pointer/RawPositionValues[14]
//     Term 20 (AT2000-0250)/Term 21 (AT2000-5250)/FB Inputs/Value Channel 16 <-> Data Pointer/RawPositionValues[15]
//     Term 20 (AT2000-0250)/Term 21 (AT2000-5250)/FB Inputs/Value Channel 17 <-> Data Pointer/RawPositionValues[16]
//     Term 20 (AT2000-0250)/Term 21 (AT2000-5250)/FB Inputs/Value Channel 18 <-> Data Pointer/RawPositionValues[17]
//     Term 20 (AT2000-0250)/Term 21 (AT2000-5250)/FB Inputs/Value Channel 19 <-> Data Pointer/RawPositionValues[18]
//     Term 20 (AT2000-0250)/Term 21 (AT2000-5250)/FB Inputs/Value Channel 20 <-> Data Pointer/RawPositionValues[19]
//     Term 20 (AT2000-0250)/Term 21 (AT2000-5250)/FB Inputs/Value Channel 21 <-> Data Pointer/RawPositionValues[20]
//     Term 20 (AT2000-0250)/Term 21 (AT2000-5250)/FB Inputs/Value Channel 22 <-> Data Pointer/RawPositionValues[21]
//     Term 20 (AT2000-0250)/Term 21 (AT2000-5250)/FB Inputs/Value Channel 23 <-> Data Pointer/RawPositionValues[22]
//     Term 20 (AT2000-0250)/Term 21 (AT2000-5250)/FB Inputs/Value Channel 24 <-> Data Pointer/RawPositionValues[23]
//     Term 20 (AT2000-0250)/Term 21 (AT2000-5250)/FB Inputs/Value Channel 25 <-> Data Pointer/RawPositionValues[24]
//     Term 20 (AT2000-0250)/Term 21 (AT2000-5250)/FB Inputs/Value Channel 26 <-> Data Pointer/RawPositionValues[25]
//     Term 20 (AT2000-0250)/Term 21 (AT2000-5250)/FB Inputs/Value Channel 27 <-> Data Pointer/RawPositionValues[26]
//     Term 20 (AT2000-0250)/Term 21 (AT2000-5250)/FB Inputs/Value Channel 28 <-> Data Pointer/RawPositionValues[27]
//     Term 20 (AT2000-0250)/Term 21 (AT2000-5250)/FB Inputs/Value Channel 29 <-> Data Pointer/RawPositionValues[28]
//     Term 20 (AT2000-0250)/Term 21 (AT2000-5250)/FB Inputs/Value Channel 30 <-> Data Pointer/RawPositionValues[29]
//     Term 20 (AT2000-0250)/Term 21 (AT2000-5250)/FB Inputs/Value Channel 31 <-> Data Pointer/RawPositionValues[30]
//     Term 20 (AT2000-0250)/Term 21 (AT2000-5250)/FB Inputs/Value Channel 32 <-> Data Pointer/RawPositionValues[31]
//   Device 8 (EtherCAT) <-> TcCOM Objects/XtsProcessingUnit 1/Part 1/Module 10
//     Term 23 (AT2001-0250)/CC Inputs/Current actual value Ch.1 <-> Data Pointer/CurrentActualValues[0]
//     Term 23 (AT2001-0250)/CC Inputs/Current actual value Ch.10 <-> Data Pointer/CurrentActualValues[9]
//     Term 23 (AT2001-0250)/CC Inputs/Current actual value Ch.11 <-> Data Pointer/CurrentActualValues[10]
//     Term 23 (AT2001-0250)/CC Inputs/Current actual value Ch.12 <-> Data Pointer/CurrentActualValues[11]
//     Term 23 (AT2001-0250)/CC Inputs/Current actual value Ch.13 <-> Data Pointer/CurrentActualValues[12]
//     Term 23 (AT2001-0250)/CC Inputs/Current actual value Ch.14 <-> Data Pointer/CurrentActualValues[13]
//     Term 23 (AT2001-0250)/CC Inputs/Current actual value Ch.15 <-> Data Pointer/CurrentActualValues[14]
//     Term 23 (AT2001-0250)/CC Inputs/Current actual value Ch.2 <-> Data Pointer/CurrentActualValues[1]
//     Term 23 (AT2001-0250)/CC Inputs/Current actual value Ch.3 <-> Data Pointer/CurrentActualValues[2]
//     Term 23 (AT2001-0250)/CC Inputs/Current actual value Ch.4 <-> Data Pointer/CurrentActualValues[3]
//     Term 23 (AT2001-0250)/CC Inputs/Current actual value Ch.5 <-> Data Pointer/CurrentActualValues[4]
//     Term 23 (AT2001-0250)/CC Inputs/Current actual value Ch.6 <-> Data Pointer/CurrentActualValues[5]
//     Term 23 (AT2001-0250)/CC Inputs/Current actual value Ch.7 <-> Data Pointer/CurrentActualValues[6]
//     Term 23 (AT2001-0250)/CC Inputs/Current actual value Ch.8 <-> Data Pointer/CurrentActualValues[7]
//     Term 23 (AT2001-0250)/CC Inputs/Current actual value Ch.9 <-> Data Pointer/CurrentActualValues[8]
//     Term 23 (AT2001-0250)/CC Inputs/Status <-> Data Pointer/Status
//     Term 23 (AT2001-0250)/CC Outputs/Control <-> Data Pointer/Control
//     Term 23 (AT2001-0250)/CC Outputs/Current setpoint value Ch.1 <-> Data Pointer/CurrentSetpointValues[0]
//     Term 23 (AT2001-0250)/CC Outputs/Current setpoint value Ch.10 <-> Data Pointer/CurrentSetpointValues[9]
//     Term 23 (AT2001-0250)/CC Outputs/Current setpoint value Ch.11 <-> Data Pointer/CurrentSetpointValues[10]
//     Term 23 (AT2001-0250)/CC Outputs/Current setpoint value Ch.12 <-> Data Pointer/CurrentSetpointValues[11]
//     Term 23 (AT2001-0250)/CC Outputs/Current setpoint value Ch.13 <-> Data Pointer/CurrentSetpointValues[12]
//     Term 23 (AT2001-0250)/CC Outputs/Current setpoint value Ch.14 <-> Data Pointer/CurrentSetpointValues[13]
//     Term 23 (AT2001-0250)/CC Outputs/Current setpoint value Ch.15 <-> Data Pointer/CurrentSetpointValues[14]
//     Term 23 (AT2001-0250)/CC Outputs/Current setpoint value Ch.2 <-> Data Pointer/CurrentSetpointValues[1]
//     Term 23 (AT2001-0250)/CC Outputs/Current setpoint value Ch.3 <-> Data Pointer/CurrentSetpointValues[2]
//     Term 23 (AT2001-0250)/CC Outputs/Current setpoint value Ch.4 <-> Data Pointer/CurrentSetpointValues[3]
//     Term 23 (AT2001-0250)/CC Outputs/Current setpoint value Ch.5 <-> Data Pointer/CurrentSetpointValues[4]
//     Term 23 (AT2001-0250)/CC Outputs/Current setpoint value Ch.6 <-> Data Pointer/CurrentSetpointValues[5]
//     Term 23 (AT2001-0250)/CC Outputs/Current setpoint value Ch.7 <-> Data Pointer/CurrentSetpointValues[6]
//     Term 23 (AT2001-0250)/CC Outputs/Current setpoint value Ch.8 <-> Data Pointer/CurrentSetpointValues[7]
//     Term 23 (AT2001-0250)/CC Outputs/Current setpoint value Ch.9 <-> Data Pointer/CurrentSetpointValues[8]
//     Term 23 (AT2001-0250)/Term 24 (AT2001-5250)/FB Inputs/Value Channel 01 <-> Data Pointer/RawPositionValues[0]
//     Term 23 (AT2001-0250)/Term 24 (AT2001-5250)/FB Inputs/Value Channel 02 <-> Data Pointer/RawPositionValues[1]
//     Term 23 (AT2001-0250)/Term 24 (AT2001-5250)/FB Inputs/Value Channel 03 <-> Data Pointer/RawPositionValues[2]
//     Term 23 (AT2001-0250)/Term 24 (AT2001-5250)/FB Inputs/Value Channel 04 <-> Data Pointer/RawPositionValues[3]
//     Term 23 (AT2001-0250)/Term 24 (AT2001-5250)/FB Inputs/Value Channel 05 <-> Data Pointer/RawPositionValues[4]
//     Term 23 (AT2001-0250)/Term 24 (AT2001-5250)/FB Inputs/Value Channel 06 <-> Data Pointer/RawPositionValues[5]
//     Term 23 (AT2001-0250)/Term 24 (AT2001-5250)/FB Inputs/Value Channel 07 <-> Data Pointer/RawPositionValues[6]
//     Term 23 (AT2001-0250)/Term 24 (AT2001-5250)/FB Inputs/Value Channel 08 <-> Data Pointer/RawPositionValues[7]
//     Term 23 (AT2001-0250)/Term 24 (AT2001-5250)/FB Inputs/Value Channel 09 <-> Data Pointer/RawPositionValues[8]
//     Term 23 (AT2001-0250)/Term 24 (AT2001-5250)/FB Inputs/Value Channel 10 <-> Data Pointer/RawPositionValues[9]
//     Term 23 (AT2001-0250)/Term 24 (AT2001-5250)/FB Inputs/Value Channel 11 <-> Data Pointer/RawPositionValues[10]
//     Term 23 (AT2001-0250)/Term 24 (AT2001-5250)/FB Inputs/Value Channel 12 <-> Data Pointer/RawPositionValues[11]
//     Term 23 (AT2001-0250)/Term 24 (AT2001-5250)/FB Inputs/Value Channel 13 <-> Data Pointer/RawPositionValues[12]
//     Term 23 (AT2001-0250)/Term 24 (AT2001-5250)/FB Inputs/Value Channel 14 <-> Data Pointer/RawPositionValues[13]
//     Term 23 (AT2001-0250)/Term 24 (AT2001-5250)/FB Inputs/Value Channel 15 <-> Data Pointer/RawPositionValues[14]
//     Term 23 (AT2001-0250)/Term 24 (AT2001-5250)/FB Inputs/Value Channel 16 <-> Data Pointer/RawPositionValues[15]
//     Term 23 (AT2001-0250)/Term 24 (AT2001-5250)/FB Inputs/Value Channel 17 <-> Data Pointer/RawPositionValues[16]
//     Term 23 (AT2001-0250)/Term 24 (AT2001-5250)/FB Inputs/Value Channel 18 <-> Data Pointer/RawPositionValues[17]
//     Term 23 (AT2001-0250)/Term 24 (AT2001-5250)/FB Inputs/Value Channel 19 <-> Data Pointer/RawPositionValues[18]
//     Term 23 (AT2001-0250)/Term 24 (AT2001-5250)/FB Inputs/Value Channel 20 <-> Data Pointer/RawPositionValues[19]
//     Term 23 (AT2001-0250)/Term 24 (AT2001-5250)/FB Inputs/Value Channel 21 <-> Data Pointer/RawPositionValues[20]
//     Term 23 (AT2001-0250)/Term 24 (AT2001-5250)/FB Inputs/Value Channel 22 <-> Data Pointer/RawPositionValues[21]
//     Term 23 (AT2001-0250)/Term 24 (AT2001-5250)/FB Inputs/Value Channel 23 <-> Data Pointer/RawPositionValues[22]
//     Term 23 (AT2001-0250)/Term 24 (AT2001-5250)/FB Inputs/Value Channel 24 <-> Data Pointer/RawPositionValues[23]
//     Term 23 (AT2001-0250)/Term 24 (AT2001-5250)/FB Inputs/Value Channel 25 <-> Data Pointer/RawPositionValues[24]
//     Term 23 (AT2001-0250)/Term 24 (AT2001-5250)/FB Inputs/Value Channel 26 <-> Data Pointer/RawPositionValues[25]
//     Term 23 (AT2001-0250)/Term 24 (AT2001-5250)/FB Inputs/Value Channel 27 <-> Data Pointer/RawPositionValues[26]
//     Term 23 (AT2001-0250)/Term 24 (AT2001-5250)/FB Inputs/Value Channel 28 <-> Data Pointer/RawPositionValues[27]
//     Term 23 (AT2001-0250)/Term 24 (AT2001-5250)/FB Inputs/Value Channel 29 <-> Data Pointer/RawPositionValues[28]
//     Term 23 (AT2001-0250)/Term 24 (AT2001-5250)/FB Inputs/Value Channel 30 <-> Data Pointer/RawPositionValues[29]
//     Term 23 (AT2001-0250)/Term 24 (AT2001-5250)/FB Inputs/Value Channel 31 <-> Data Pointer/RawPositionValues[30]
//     Term 23 (AT2001-0250)/Term 24 (AT2001-5250)/FB Inputs/Value Channel 32 <-> Data Pointer/RawPositionValues[31]
//   Device 8 (EtherCAT) <-> TcCOM Objects/XtsProcessingUnit 1/Part 1/Module 11
//     Term 25 (AT2050-0500)/CC Inputs/Current actual value Ch.1 <-> Data Pointer/CurrentActualValues[0]
//     Term 25 (AT2050-0500)/CC Inputs/Current actual value Ch.10 <-> Data Pointer/CurrentActualValues[9]
//     Term 25 (AT2050-0500)/CC Inputs/Current actual value Ch.11 <-> Data Pointer/CurrentActualValues[10]
//     Term 25 (AT2050-0500)/CC Inputs/Current actual value Ch.12 <-> Data Pointer/CurrentActualValues[11]
//     Term 25 (AT2050-0500)/CC Inputs/Current actual value Ch.13 <-> Data Pointer/CurrentActualValues[12]
//     Term 25 (AT2050-0500)/CC Inputs/Current actual value Ch.14 <-> Data Pointer/CurrentActualValues[13]
//     Term 25 (AT2050-0500)/CC Inputs/Current actual value Ch.15 <-> Data Pointer/CurrentActualValues[14]
//     Term 25 (AT2050-0500)/CC Inputs/Current actual value Ch.2 <-> Data Pointer/CurrentActualValues[1]
//     Term 25 (AT2050-0500)/CC Inputs/Current actual value Ch.3 <-> Data Pointer/CurrentActualValues[2]
//     Term 25 (AT2050-0500)/CC Inputs/Current actual value Ch.4 <-> Data Pointer/CurrentActualValues[3]
//     Term 25 (AT2050-0500)/CC Inputs/Current actual value Ch.5 <-> Data Pointer/CurrentActualValues[4]
//     Term 25 (AT2050-0500)/CC Inputs/Current actual value Ch.6 <-> Data Pointer/CurrentActualValues[5]
//     Term 25 (AT2050-0500)/CC Inputs/Current actual value Ch.7 <-> Data Pointer/CurrentActualValues[6]
//     Term 25 (AT2050-0500)/CC Inputs/Current actual value Ch.8 <-> Data Pointer/CurrentActualValues[7]
//     Term 25 (AT2050-0500)/CC Inputs/Current actual value Ch.9 <-> Data Pointer/CurrentActualValues[8]
//     Term 25 (AT2050-0500)/CC Inputs/Status <-> Data Pointer/Status
//     Term 25 (AT2050-0500)/CC Outputs/Control <-> Data Pointer/Control
//     Term 25 (AT2050-0500)/CC Outputs/Current setpoint value Ch.1 <-> Data Pointer/CurrentSetpointValues[0]
//     Term 25 (AT2050-0500)/CC Outputs/Current setpoint value Ch.10 <-> Data Pointer/CurrentSetpointValues[9]
//     Term 25 (AT2050-0500)/CC Outputs/Current setpoint value Ch.11 <-> Data Pointer/CurrentSetpointValues[10]
//     Term 25 (AT2050-0500)/CC Outputs/Current setpoint value Ch.12 <-> Data Pointer/CurrentSetpointValues[11]
//     Term 25 (AT2050-0500)/CC Outputs/Current setpoint value Ch.13 <-> Data Pointer/CurrentSetpointValues[12]
//     Term 25 (AT2050-0500)/CC Outputs/Current setpoint value Ch.14 <-> Data Pointer/CurrentSetpointValues[13]
//     Term 25 (AT2050-0500)/CC Outputs/Current setpoint value Ch.15 <-> Data Pointer/CurrentSetpointValues[14]
//     Term 25 (AT2050-0500)/CC Outputs/Current setpoint value Ch.2 <-> Data Pointer/CurrentSetpointValues[1]
//     Term 25 (AT2050-0500)/CC Outputs/Current setpoint value Ch.3 <-> Data Pointer/CurrentSetpointValues[2]
//     Term 25 (AT2050-0500)/CC Outputs/Current setpoint value Ch.4 <-> Data Pointer/CurrentSetpointValues[3]
//     Term 25 (AT2050-0500)/CC Outputs/Current setpoint value Ch.5 <-> Data Pointer/CurrentSetpointValues[4]
//     Term 25 (AT2050-0500)/CC Outputs/Current setpoint value Ch.6 <-> Data Pointer/CurrentSetpointValues[5]
//     Term 25 (AT2050-0500)/CC Outputs/Current setpoint value Ch.7 <-> Data Pointer/CurrentSetpointValues[6]
//     Term 25 (AT2050-0500)/CC Outputs/Current setpoint value Ch.8 <-> Data Pointer/CurrentSetpointValues[7]
//     Term 25 (AT2050-0500)/CC Outputs/Current setpoint value Ch.9 <-> Data Pointer/CurrentSetpointValues[8]
//     Term 25 (AT2050-0500)/Term 26 (AT2050-5500)/FB Inputs/Value Channel 01 <-> Data Pointer/RawPositionValues[0]
//     Term 25 (AT2050-0500)/Term 26 (AT2050-5500)/FB Inputs/Value Channel 02 <-> Data Pointer/RawPositionValues[1]
//     Term 25 (AT2050-0500)/Term 26 (AT2050-5500)/FB Inputs/Value Channel 03 <-> Data Pointer/RawPositionValues[2]
//     Term 25 (AT2050-0500)/Term 26 (AT2050-5500)/FB Inputs/Value Channel 04 <-> Data Pointer/RawPositionValues[3]
//     Term 25 (AT2050-0500)/Term 26 (AT2050-5500)/FB Inputs/Value Channel 05 <-> Data Pointer/RawPositionValues[4]
//     Term 25 (AT2050-0500)/Term 26 (AT2050-5500)/FB Inputs/Value Channel 06 <-> Data Pointer/RawPositionValues[5]
//     Term 25 (AT2050-0500)/Term 26 (AT2050-5500)/FB Inputs/Value Channel 07 <-> Data Pointer/RawPositionValues[6]
//     Term 25 (AT2050-0500)/Term 26 (AT2050-5500)/FB Inputs/Value Channel 08 <-> Data Pointer/RawPositionValues[7]
//     Term 25 (AT2050-0500)/Term 26 (AT2050-5500)/FB Inputs/Value Channel 09 <-> Data Pointer/RawPositionValues[8]
//     Term 25 (AT2050-0500)/Term 26 (AT2050-5500)/FB Inputs/Value Channel 10 <-> Data Pointer/RawPositionValues[9]
//     Term 25 (AT2050-0500)/Term 26 (AT2050-5500)/FB Inputs/Value Channel 11 <-> Data Pointer/RawPositionValues[10]
//     Term 25 (AT2050-0500)/Term 26 (AT2050-5500)/FB Inputs/Value Channel 12 <-> Data Pointer/RawPositionValues[11]
//     Term 25 (AT2050-0500)/Term 26 (AT2050-5500)/FB Inputs/Value Channel 13 <-> Data Pointer/RawPositionValues[12]
//     Term 25 (AT2050-0500)/Term 26 (AT2050-5500)/FB Inputs/Value Channel 14 <-> Data Pointer/RawPositionValues[13]
//     Term 25 (AT2050-0500)/Term 26 (AT2050-5500)/FB Inputs/Value Channel 15 <-> Data Pointer/RawPositionValues[14]
//     Term 25 (AT2050-0500)/Term 26 (AT2050-5500)/FB Inputs/Value Channel 16 <-> Data Pointer/RawPositionValues[15]
//     Term 25 (AT2050-0500)/Term 26 (AT2050-5500)/FB Inputs/Value Channel 17 <-> Data Pointer/RawPositionValues[16]
//     Term 25 (AT2050-0500)/Term 26 (AT2050-5500)/FB Inputs/Value Channel 18 <-> Data Pointer/RawPositionValues[17]
//     Term 25 (AT2050-0500)/Term 26 (AT2050-5500)/FB Inputs/Value Channel 19 <-> Data Pointer/RawPositionValues[18]
//     Term 25 (AT2050-0500)/Term 26 (AT2050-5500)/FB Inputs/Value Channel 20 <-> Data Pointer/RawPositionValues[19]
//     Term 25 (AT2050-0500)/Term 26 (AT2050-5500)/FB Inputs/Value Channel 21 <-> Data Pointer/RawPositionValues[20]
//     Term 25 (AT2050-0500)/Term 26 (AT2050-5500)/FB Inputs/Value Channel 22 <-> Data Pointer/RawPositionValues[21]
//     Term 25 (AT2050-0500)/Term 26 (AT2050-5500)/FB Inputs/Value Channel 23 <-> Data Pointer/RawPositionValues[22]
//     Term 25 (AT2050-0500)/Term 26 (AT2050-5500)/FB Inputs/Value Channel 24 <-> Data Pointer/RawPositionValues[23]
//     Term 25 (AT2050-0500)/Term 26 (AT2050-5500)/FB Inputs/Value Channel 25 <-> Data Pointer/RawPositionValues[24]
//     Term 25 (AT2050-0500)/Term 26 (AT2050-5500)/FB Inputs/Value Channel 26 <-> Data Pointer/RawPositionValues[25]
//     Term 25 (AT2050-0500)/Term 26 (AT2050-5500)/FB Inputs/Value Channel 27 <-> Data Pointer/RawPositionValues[26]
//     Term 25 (AT2050-0500)/Term 26 (AT2050-5500)/FB Inputs/Value Channel 28 <-> Data Pointer/RawPositionValues[27]
//     Term 25 (AT2050-0500)/Term 26 (AT2050-5500)/FB Inputs/Value Channel 29 <-> Data Pointer/RawPositionValues[28]
//     Term 25 (AT2050-0500)/Term 26 (AT2050-5500)/FB Inputs/Value Channel 30 <-> Data Pointer/RawPositionValues[29]
//     Term 25 (AT2050-0500)/Term 26 (AT2050-5500)/FB Inputs/Value Channel 31 <-> Data Pointer/RawPositionValues[30]
//     Term 25 (AT2050-0500)/Term 26 (AT2050-5500)/FB Inputs/Value Channel 32 <-> Data Pointer/RawPositionValues[31]
//   Device 8 (EtherCAT) <-> TcCOM Objects/XtsProcessingUnit 1/Part 1/Module 12
//     Term 27 (AT2050-0501)/CC Inputs/Current actual value Ch.1 <-> Data Pointer/CurrentActualValues[0]
//     Term 27 (AT2050-0501)/CC Inputs/Current actual value Ch.10 <-> Data Pointer/CurrentActualValues[9]
//     Term 27 (AT2050-0501)/CC Inputs/Current actual value Ch.11 <-> Data Pointer/CurrentActualValues[10]
//     Term 27 (AT2050-0501)/CC Inputs/Current actual value Ch.12 <-> Data Pointer/CurrentActualValues[11]
//     Term 27 (AT2050-0501)/CC Inputs/Current actual value Ch.13 <-> Data Pointer/CurrentActualValues[12]
//     Term 27 (AT2050-0501)/CC Inputs/Current actual value Ch.14 <-> Data Pointer/CurrentActualValues[13]
//     Term 27 (AT2050-0501)/CC Inputs/Current actual value Ch.15 <-> Data Pointer/CurrentActualValues[14]
//     Term 27 (AT2050-0501)/CC Inputs/Current actual value Ch.2 <-> Data Pointer/CurrentActualValues[1]
//     Term 27 (AT2050-0501)/CC Inputs/Current actual value Ch.3 <-> Data Pointer/CurrentActualValues[2]
//     Term 27 (AT2050-0501)/CC Inputs/Current actual value Ch.4 <-> Data Pointer/CurrentActualValues[3]
//     Term 27 (AT2050-0501)/CC Inputs/Current actual value Ch.5 <-> Data Pointer/CurrentActualValues[4]
//     Term 27 (AT2050-0501)/CC Inputs/Current actual value Ch.6 <-> Data Pointer/CurrentActualValues[5]
//     Term 27 (AT2050-0501)/CC Inputs/Current actual value Ch.7 <-> Data Pointer/CurrentActualValues[6]
//     Term 27 (AT2050-0501)/CC Inputs/Current actual value Ch.8 <-> Data Pointer/CurrentActualValues[7]
//     Term 27 (AT2050-0501)/CC Inputs/Current actual value Ch.9 <-> Data Pointer/CurrentActualValues[8]
//     Term 27 (AT2050-0501)/CC Inputs/Status <-> Data Pointer/Status
//     Term 27 (AT2050-0501)/CC Outputs/Control <-> Data Pointer/Control
//     Term 27 (AT2050-0501)/CC Outputs/Current setpoint value Ch.1 <-> Data Pointer/CurrentSetpointValues[0]
//     Term 27 (AT2050-0501)/CC Outputs/Current setpoint value Ch.10 <-> Data Pointer/CurrentSetpointValues[9]
//     Term 27 (AT2050-0501)/CC Outputs/Current setpoint value Ch.11 <-> Data Pointer/CurrentSetpointValues[10]
//     Term 27 (AT2050-0501)/CC Outputs/Current setpoint value Ch.12 <-> Data Pointer/CurrentSetpointValues[11]
//     Term 27 (AT2050-0501)/CC Outputs/Current setpoint value Ch.13 <-> Data Pointer/CurrentSetpointValues[12]
//     Term 27 (AT2050-0501)/CC Outputs/Current setpoint value Ch.14 <-> Data Pointer/CurrentSetpointValues[13]
//     Term 27 (AT2050-0501)/CC Outputs/Current setpoint value Ch.15 <-> Data Pointer/CurrentSetpointValues[14]
//     Term 27 (AT2050-0501)/CC Outputs/Current setpoint value Ch.2 <-> Data Pointer/CurrentSetpointValues[1]
//     Term 27 (AT2050-0501)/CC Outputs/Current setpoint value Ch.3 <-> Data Pointer/CurrentSetpointValues[2]
//     Term 27 (AT2050-0501)/CC Outputs/Current setpoint value Ch.4 <-> Data Pointer/CurrentSetpointValues[3]
//     Term 27 (AT2050-0501)/CC Outputs/Current setpoint value Ch.5 <-> Data Pointer/CurrentSetpointValues[4]
//     Term 27 (AT2050-0501)/CC Outputs/Current setpoint value Ch.6 <-> Data Pointer/CurrentSetpointValues[5]
//     Term 27 (AT2050-0501)/CC Outputs/Current setpoint value Ch.7 <-> Data Pointer/CurrentSetpointValues[6]
//     Term 27 (AT2050-0501)/CC Outputs/Current setpoint value Ch.8 <-> Data Pointer/CurrentSetpointValues[7]
//     Term 27 (AT2050-0501)/CC Outputs/Current setpoint value Ch.9 <-> Data Pointer/CurrentSetpointValues[8]
//     Term 27 (AT2050-0501)/Term 28 (AT2050-5501)/FB Inputs/Value Channel 01 <-> Data Pointer/RawPositionValues[0]
//     Term 27 (AT2050-0501)/Term 28 (AT2050-5501)/FB Inputs/Value Channel 02 <-> Data Pointer/RawPositionValues[1]
//     Term 27 (AT2050-0501)/Term 28 (AT2050-5501)/FB Inputs/Value Channel 03 <-> Data Pointer/RawPositionValues[2]
//     Term 27 (AT2050-0501)/Term 28 (AT2050-5501)/FB Inputs/Value Channel 04 <-> Data Pointer/RawPositionValues[3]
//     Term 27 (AT2050-0501)/Term 28 (AT2050-5501)/FB Inputs/Value Channel 05 <-> Data Pointer/RawPositionValues[4]
//     Term 27 (AT2050-0501)/Term 28 (AT2050-5501)/FB Inputs/Value Channel 06 <-> Data Pointer/RawPositionValues[5]
//     Term 27 (AT2050-0501)/Term 28 (AT2050-5501)/FB Inputs/Value Channel 07 <-> Data Pointer/RawPositionValues[6]
//     Term 27 (AT2050-0501)/Term 28 (AT2050-5501)/FB Inputs/Value Channel 08 <-> Data Pointer/RawPositionValues[7]
//     Term 27 (AT2050-0501)/Term 28 (AT2050-5501)/FB Inputs/Value Channel 09 <-> Data Pointer/RawPositionValues[8]
//     Term 27 (AT2050-0501)/Term 28 (AT2050-5501)/FB Inputs/Value Channel 10 <-> Data Pointer/RawPositionValues[9]
//     Term 27 (AT2050-0501)/Term 28 (AT2050-5501)/FB Inputs/Value Channel 11 <-> Data Pointer/RawPositionValues[10]
//     Term 27 (AT2050-0501)/Term 28 (AT2050-5501)/FB Inputs/Value Channel 12 <-> Data Pointer/RawPositionValues[11]
//     Term 27 (AT2050-0501)/Term 28 (AT2050-5501)/FB Inputs/Value Channel 13 <-> Data Pointer/RawPositionValues[12]
//     Term 27 (AT2050-0501)/Term 28 (AT2050-5501)/FB Inputs/Value Channel 14 <-> Data Pointer/RawPositionValues[13]
//     Term 27 (AT2050-0501)/Term 28 (AT2050-5501)/FB Inputs/Value Channel 15 <-> Data Pointer/RawPositionValues[14]
//     Term 27 (AT2050-0501)/Term 28 (AT2050-5501)/FB Inputs/Value Channel 16 <-> Data Pointer/RawPositionValues[15]
//     Term 27 (AT2050-0501)/Term 28 (AT2050-5501)/FB Inputs/Value Channel 17 <-> Data Pointer/RawPositionValues[16]
//     Term 27 (AT2050-0501)/Term 28 (AT2050-5501)/FB Inputs/Value Channel 18 <-> Data Pointer/RawPositionValues[17]
//     Term 27 (AT2050-0501)/Term 28 (AT2050-5501)/FB Inputs/Value Channel 19 <-> Data Pointer/RawPositionValues[18]
//     Term 27 (AT2050-0501)/Term 28 (AT2050-5501)/FB Inputs/Value Channel 20 <-> Data Pointer/RawPositionValues[19]
//     Term 27 (AT2050-0501)/Term 28 (AT2050-5501)/FB Inputs/Value Channel 21 <-> Data Pointer/RawPositionValues[20]
//     Term 27 (AT2050-0501)/Term 28 (AT2050-5501)/FB Inputs/Value Channel 22 <-> Data Pointer/RawPositionValues[21]
//     Term 27 (AT2050-0501)/Term 28 (AT2050-5501)/FB Inputs/Value Channel 23 <-> Data Pointer/RawPositionValues[22]
//     Term 27 (AT2050-0501)/Term 28 (AT2050-5501)/FB Inputs/Value Channel 24 <-> Data Pointer/RawPositionValues[23]
//     Term 27 (AT2050-0501)/Term 28 (AT2050-5501)/FB Inputs/Value Channel 25 <-> Data Pointer/RawPositionValues[24]
//     Term 27 (AT2050-0501)/Term 28 (AT2050-5501)/FB Inputs/Value Channel 26 <-> Data Pointer/RawPositionValues[25]
//     Term 27 (AT2050-0501)/Term 28 (AT2050-5501)/FB Inputs/Value Channel 27 <-> Data Pointer/RawPositionValues[26]
//     Term 27 (AT2050-0501)/Term 28 (AT2050-5501)/FB Inputs/Value Channel 28 <-> Data Pointer/RawPositionValues[27]
//     Term 27 (AT2050-0501)/Term 28 (AT2050-5501)/FB Inputs/Value Channel 29 <-> Data Pointer/RawPositionValues[28]
//     Term 27 (AT2050-0501)/Term 28 (AT2050-5501)/FB Inputs/Value Channel 30 <-> Data Pointer/RawPositionValues[29]
//     Term 27 (AT2050-0501)/Term 28 (AT2050-5501)/FB Inputs/Value Channel 31 <-> Data Pointer/RawPositionValues[30]
//     Term 27 (AT2050-0501)/Term 28 (AT2050-5501)/FB Inputs/Value Channel 32 <-> Data Pointer/RawPositionValues[31]
//   NC-Task 1 SAF/Axes/Mover Axis 1 <-> TcCOM Objects/XtsProcessingUnit 1/Mover 1
//     SoftDrive 1/Data Pointer/InputPointer1 <-> Inputs/SoftDriveInput
//     SoftDrive 1/Data Pointer/OutputPointer1 <-> Outputs/SoftDriveOutput
//   NC-Task 1 SAF/Axes/Mover Axis 2 <-> TcCOM Objects/XtsProcessingUnit 1/Mover 2
//     SoftDrive 2/Data Pointer/InputPointer1 <-> Inputs/SoftDriveInput
//     SoftDrive 2/Data Pointer/OutputPointer1 <-> Outputs/SoftDriveOutput
//   NC-Task 1 SAF/Axes/Mover Axis 3 <-> TcCOM Objects/XtsProcessingUnit 1/Mover 3
//     SoftDrive 3/Data Pointer/InputPointer1 <-> Inputs/SoftDriveInput
//     SoftDrive 3/Data Pointer/OutputPointer1 <-> Outputs/SoftDriveOutput
//   NC-Task 1 SAF/Axes/Mover Axis 4 <-> TcCOM Objects/XtsProcessingUnit 1/Mover 4
//     SoftDrive 4/Data Pointer/InputPointer1 <-> Inputs/SoftDriveInput
//     SoftDrive 4/Data Pointer/OutputPointer1 <-> Outputs/SoftDriveOutput
//   NC-Task 1 SAF/Axes/Mover Axis 5 <-> TcCOM Objects/XtsProcessingUnit 1/Mover 5
//     SoftDrive 5/Data Pointer/InputPointer1 <-> Inputs/SoftDriveInput
//     SoftDrive 5/Data Pointer/OutputPointer1 <-> Outputs/SoftDriveOutput
//   NC-Task 1 SAF/Axes/Mover Axis 6 <-> TcCOM Objects/XtsProcessingUnit 1/Mover 6
//     SoftDrive 6/Data Pointer/InputPointer1 <-> Inputs/SoftDriveInput
//     SoftDrive 6/Data Pointer/OutputPointer1 <-> Outputs/SoftDriveOutput
//   NC-Task 1 SAF/Axes/Mover Axis 7 <-> TcCOM Objects/XtsProcessingUnit 1/Mover 7
//     SoftDrive 7/Data Pointer/InputPointer1 <-> Inputs/SoftDriveInput
//     SoftDrive 7/Data Pointer/OutputPointer1 <-> Outputs/SoftDriveOutput
//   NC-Task 1 SAF/Axes/Mover Axis 8 <-> TcCOM Objects/XtsProcessingUnit 1/Mover 8
//     SoftDrive 8/Data Pointer/InputPointer1 <-> Inputs/SoftDriveInput
//     SoftDrive 8/Data Pointer/OutputPointer1 <-> Outputs/SoftDriveOutput
//   Plc/Plc Instance <-> NC-Task 1 SAF/Axes/Mover Axis 1
//     PlcTask Inputs/MAIN.aMovers[1].Axis.Axis.NcToPlc <-> Outputs/ToPlc
//     PlcTask Outputs/MAIN.aMovers[1].Axis.Axis.PlcToNc <-> Inputs/FromPlc
//   Plc/Plc Instance <-> NC-Task 1 SAF/Axes/Mover Axis 2
//     PlcTask Inputs/MAIN.aMovers[2].Axis.Axis.NcToPlc <-> Outputs/ToPlc
//     PlcTask Outputs/MAIN.aMovers[2].Axis.Axis.PlcToNc <-> Inputs/FromPlc
//   Plc/Plc Instance <-> NC-Task 1 SAF/Axes/Mover Axis 3
//     PlcTask Inputs/MAIN.aMovers[3].Axis.Axis.NcToPlc <-> Outputs/ToPlc
//     PlcTask Outputs/MAIN.aMovers[3].Axis.Axis.PlcToNc <-> Inputs/FromPlc
//   Plc/Plc Instance <-> NC-Task 1 SAF/Axes/Mover Axis 4
//     PlcTask Inputs/MAIN.aMovers[4].Axis.Axis.NcToPlc <-> Outputs/ToPlc
//     PlcTask Outputs/MAIN.aMovers[4].Axis.Axis.PlcToNc <-> Inputs/FromPlc
//   Plc/Plc Instance <-> NC-Task 1 SAF/Axes/Mover Axis 5
//     PlcTask Inputs/MAIN.aMovers[5].Axis.Axis.NcToPlc <-> Outputs/ToPlc
//     PlcTask Outputs/MAIN.aMovers[5].Axis.Axis.PlcToNc <-> Inputs/FromPlc
//   Plc/Plc Instance <-> NC-Task 1 SAF/Axes/Mover Axis 6
